gfCNCPoint1[28798] = {X 213.7862, Y 102.3021, Z -2.1667, A 0.000, B 0.000, C 0.000 }
gfCNCPoint1[28799] = {X 213.3966, Y 102.2485, Z -2.1667, A 0.000, B 0.000, C 0.000 }
gfCNCPoint1[28800] = {X 213.0070, Y 102.3021, Z -2.1667, A 0.000, B 0.000, C 0.000 }
gfCNCPoint1[28801] = {X 212.6141, Y 102.3200, Z -2.1667, A 0.000, B 0.000, C 0.000 }
gfCNCPoint1[28802] = {X 194.9870, Y 102.3200, Z -2.1667, A 0.000, B 0.000, C 0.000 }
gfCNCPoint1[28803] = {X 194.0257, Y 102.2117, Z -2.1667, A 0.000, B 0.000, C 0.000 }
gfCNCPoint1[28804] = {X 193.1126, Y 101.8922, Z -2.1667, A 0.000, B 0.000, C 0.000 }
gfCNCPoint1[28805] = {X 192.2935, Y 101.3775, Z -2.1667, A 0.000, B 0.000, C 0.000 }
gfCNCPoint1[28806] = {X 191.6094, Y 100.6935, Z -2.1667, A 0.000, B 0.000, C 0.000 }
gfCNCPoint1[28807] = {X 191.0948, Y 99.8744, Z -2.1667, A 0.000, B 0.000, C 0.000 }
gfCNCPoint1[28808] = {X 190.7753, Y 98.9613, Z -2.1667, A 0.000, B 0.000, C 0.000 }
gfCNCPoint1[28809] = {X 190.6670, Y 98.0000, Z -2.1667, A 0.000, B 0.000, C 0.000 }
gfCNCPoint1[28810] = {X 190.6670, Y 97.0659, Z -2.1667, A 0.000, B 0.000, C 0.000 }
gfCNCPoint1[28811] = {X 190.7727, Y 96.1162, Z -2.1667, A 0.000, B 0.000, C 0.000 }
gfCNCPoint1[28812] = {X 191.0846, Y 95.2129, Z -2.1667, A 0.000, B 0.000, C 0.000 }
gfCNCPoint1[28813] = {X 191.5874, Y 94.4003, Z -2.1667, A 0.000, B 0.000, C 0.000 }
gfCNCPoint1[28814] = {X 188.5647, Y 91.1002, Z -2.1667, A 0.000, B 0.000, C 0.000 }
gfCNCPoint1[28815] = {X 150.0898, Y 91.1002, Z -2.1667, A 0.000, B 0.000, C 0.000 }
gfCNCPoint1[28816] = {X 147.1445, Y 94.3633, Z -2.1667, A 0.000, B 0.000, C 0.000 }
gfCNCPoint1[28817] = {X 147.6631, Y 95.1844, Z -2.1667, A 0.000, B 0.000, C 0.000 }
gfCNCPoint1[28818] = {X 147.9867, Y 96.1001, Z -2.1667, A 0.000, B 0.000, C 0.000 }
gfCNCPoint1[28819] = {X 148.0991, Y 97.0648, Z -2.1667, A 0.000, B 0.000, C 0.000 }
gfCNCPoint1[28820] = {X 148.0991, Y 98.0000, Z -2.1667, A 0.000, B 0.000, C 0.000 }
gfCNCPoint1[28821] = {X 147.9908, Y 98.9613, Z -2.1667, A 0.000, B 0.000, C 0.000 }
gfCNCPoint1[28822] = {X 147.6713, Y 99.8744, Z -2.1667, A 0.000, B 0.000, C 0.000 }
gfCNCPoint1[28823] = {X 147.1566, Y 100.6935, Z -2.1667, A 0.000, B 0.000, C 0.000 }
gfCNCPoint1[28824] = {X 146.4726, Y 101.3775, Z -2.1667, A 0.000, B 0.000, C 0.000 }
gfCNCPoint1[28825] = {X 145.6535, Y 101.8922, Z -2.1667, A 0.000, B 0.000, C 0.000 }
gfCNCPoint1[28826] = {X 144.7404, Y 102.2117, Z -2.1667, A 0.000, B 0.000, C 0.000 }
gfCNCPoint1[28827] = {X 143.7791, Y 102.3200, Z -2.1667, A 0.000, B 0.000, C 0.000 }
gfCNCPoint1[28828] = {X 125.0000, Y 102.3200, Z -2.1667, A 0.000, B 0.000, C 0.000 }
gfCNCPoint1[28829] = {X 124.0387, Y 102.2117, Z -2.1667, A 0.000, B 0.000, C 0.000 }
gfCNCPoint1[28830] = {X 123.1256, Y 101.8922, Z -2.1667, A 0.000, B 0.000, C 0.000 }
gfCNCPoint1[28831] = {X 122.3065, Y 101.3775, Z -2.1667, A 0.000, B 0.000, C 0.000 }
gfCNCPoint1[28832] = {X 121.6225, Y 100.6935, Z -2.1667, A 0.000, B 0.000, C 0.000 }
gfCNCPoint1[28833] = {X 121.1078, Y 99.8744, Z -2.1667, A 0.000, B 0.000, C 0.000 }
gfCNCPoint1[28834] = {X 120.7883, Y 98.9613, Z -2.1667, A 0.000, B 0.000, C 0.000 }
gfCNCPoint1[28835] = {X 120.6800, Y 98.0000, Z -2.1667, A 0.000, B 0.000, C 0.000 }
gfCNCPoint1[28836] = {X 120.6800, Y 97.0659, Z -2.1667, A 0.000, B 0.000, C 0.000 }
gfCNCPoint1[28837] = {X 120.7833, Y 96.1270, Z -2.1667, A 0.000, B 0.000, C 0.000 }
gfCNCPoint1[28838] = {X 121.0882, Y 95.2329, Z -2.1667, A 0.000, B 0.000, C 0.000 }
gfCNCPoint1[28839] = {X 121.5801, Y 94.4265, Z -2.1667, A 0.000, B 0.000, C 0.000 }
gfCNCPoint1[28840] = {X 122.2355, Y 93.7463, Z -2.1667, A 0.000, B 0.000, C 0.000 }
gfCNCPoint1[28841] = {X 123.0231, Y 93.2248, Z -2.1667, A 0.000, B 0.000, C 0.000 }
gfCNCPoint1[28842] = {X 123.9052, Y 92.8870, Z -2.1667, A 0.000, B 0.000, C 0.000 }
gfCNCPoint1[28843] = {X 124.8397, Y 92.7489, Z -2.1667, A 0.000, B 0.000, C 0.000 }
gfCNCPoint1[28844] = {X 124.8829, Y 92.7325, Z -2.1667, A 0.000, B 0.000, C 0.000 }
gfCNCPoint1[28845] = {X 124.9280, Y 92.7225, Z -2.1667, A 0.000, B 0.000, C 0.000 }
gfCNCPoint1[28846] = {X 125.4501, Y 92.6450, Z -2.1667, A 0.000, B 0.000, C 0.000 }
gfCNCPoint1[28847] = {X 126.2811, Y 92.5043, Z -2.1667, A 0.000, B 0.000, C 0.000 }
gfCNCPoint1[28848] = {X 127.1008, Y 92.3085, Z -2.1667, A 0.000, B 0.000, C 0.000 }
gfCNCPoint1[28849] = {X 128.3225, Y 91.1566, Z -2.1667, A 0.000, B 0.000, C 0.000 }
gfCNCPoint1[28850] = {X 129.4799, Y 89.9402, Z -2.1667, A 0.000, B 0.000, C 0.000 }
gfCNCPoint1[28851] = {X 140.6805, Y 77.6405, Z -2.1667, A 0.000, B 0.000, C 0.000 }
gfCNCPoint1[28852] = {X 137.7230, Y 74.9473, Z -2.1667, A 0.000, B 0.000, C 0.000 }
gfCNCPoint1[28853] = {X 140.7396, Y 77.6944, Z -2.1667, A 0.000, B 0.000, C 0.000 }
gfCNCPoint1[28854] = {X 155.7331, Y 61.2296, Z -2.1667, A 0.000, B 0.000, C 0.000 }
gfCNCPoint1[28855] = {X 155.3670, Y 60.5231, Z -2.1667, A 0.000, B 0.000, C 0.000 }
gfCNCPoint1[28856] = {X 155.1393, Y 59.7606, Z -2.1667, A 0.000, B 0.000, C 0.000 }
gfCNCPoint1[28857] = {X 155.0581, Y 58.9691, Z -2.1667, A 0.000, B 0.000, C 0.000 }
gfCNCPoint1[28858] = {X 155.0580, Y 58.0000, Z -2.1667, A 0.000, B 0.000, C 0.000 }
gfCNCPoint1[28859] = {X 155.1643, Y 57.0565, Z -2.1667, A 0.000, B 0.000, C 0.000 }
gfCNCPoint1[28860] = {X 155.4778, Y 56.1603, Z -2.1667, A 0.000, B 0.000, C 0.000 }
gfCNCPoint1[28861] = {X 155.9830, Y 55.3564, Z -2.1667, A 0.000, B 0.000, C 0.000 }
gfCNCPoint1[28862] = {X 156.6544, Y 54.6850, Z -2.1667, A 0.000, B 0.000, C 0.000 }
gfCNCPoint1[28863] = {X 157.4583, Y 54.1799, Z -2.1667, A 0.000, B 0.000, C 0.000 }
gfCNCPoint1[28864] = {X 158.3545, Y 53.8663, Z -2.1667, A 0.000, B 0.000, C 0.000 }
gfCNCPoint1[28865] = {X 159.2980, Y 53.7600, Z -2.1667, A 0.000, B 0.000, C 0.000 }
gfCNCPoint1[28866] = {X 178.5335, Y 53.7600, Z -2.1667, A 0.000, B 0.000, C 0.000 }
gfCNCPoint1[28867] = {X 179.4770, Y 53.8663, Z -2.1667, A 0.000, B 0.000, C 0.000 }
gfCNCPoint1[28868] = {X 180.3732, Y 54.1799, Z -2.1667, A 0.000, B 0.000, C 0.000 }
gfCNCPoint1[28869] = {X 181.1771, Y 54.6850, Z -2.1667, A 0.000, B 0.000, C 0.000 }
gfCNCPoint1[28870] = {X 181.8485, Y 55.3564, Z -2.1667, A 0.000, B 0.000, C 0.000 }
gfCNCPoint1[28871] = {X 182.3536, Y 56.1603, Z -2.1667, A 0.000, B 0.000, C 0.000 }
gfCNCPoint1[28872] = {X 182.6672, Y 57.0565, Z -2.1667, A 0.000, B 0.000, C 0.000 }
gfCNCPoint1[28873] = {X 182.7735, Y 58.0000, Z -2.1667, A 0.000, B 0.000, C 0.000 }
gfCNCPoint1[28874] = {X 182.7735, Y 58.9342, Z -2.1667, A 0.000, B 0.000, C 0.000 }
gfCNCPoint1[28875] = {X 182.6984, Y 59.7287, Z -2.1667, A 0.000, B 0.000, C 0.000 }
gfCNCPoint1[28876] = {X 182.4757, Y 60.4950, Z -2.1667, A 0.000, B 0.000, C 0.000 }
gfCNCPoint1[28877] = {X 182.1134, Y 61.2060, Z -2.1667, A 0.000, B 0.000, C 0.000 }
gfCNCPoint1[28878] = {X 209.4186, Y 91.0079, Z -2.1667, A 0.000, B 0.000, C 0.000 }
gfCNCPoint1[28879] = {X 210.0808, Y 91.6798, Z -2.1667, A 0.000, B 0.000, C 0.000 }
gfCNCPoint1[28880] = {X 210.7901, Y 92.3017, Z -2.1667, A 0.000, B 0.000, C 0.000 }
gfCNCPoint1[28881] = {X 211.0808, Y 92.4854, Z -2.1667, A 0.000, B 0.000, C 0.000 }
gfCNCPoint1[28882] = {X 211.4066, Y 92.5950, Z -2.1667, A 0.000, B 0.000, C 0.000 }
gfCNCPoint1[28883] = {X 213.4016, Y 92.9061, Z -2.1667, A 0.000, B 0.000, C 0.000 }
gfCNCPoint1[28884] = {X 214.4545, Y 92.8170, Z -2.1667, A 0.000, B 0.000, C 0.000 }
gfCNCPoint1[28885] = {X 215.5096, Y 92.7565, Z -2.1667, A 0.000, B 0.000, C 0.000 }
gfCNCPoint1[28886] = {X 216.1940, Y 92.6814, Z -2.1667, A 0.000, B 0.000, C 0.000 }
gfCNCPoint1[28887] = {X 216.8530, Y 92.4820, Z -2.1667, A 0.000, B 0.000, C 0.000 }
gfCNCPoint1[28888] = {X 217.4644, Y 92.1653, Z -2.1667, A 0.000, B 0.000, C 0.000 }
gfCNCPoint1[28889] = {X 223.0046, Y 88.5899, Z -2.1667, A 0.000, B 0.000, C 0.000 }
gfCNCPoint1[28890] = {X 246.0044, Y 73.8823, Z -2.1667, A 0.000, B 0.000, C 0.000 }
gfCNCPoint1[28891] = {X 221.6602, Y 64.3284, Z -2.1667, A 0.000, B 0.000, C 0.000 }
gfCNCPoint1[28892] = {X 219.8842, Y 63.7340, Z -2.1667, A 0.000, B 0.000, C 0.000 }
gfCNCPoint1[28893] = {X 218.0518, Y 63.3467, Z -2.1667, A 0.000, B 0.000, C 0.000 }
gfCNCPoint1[28894] = {X 216.1871, Y 63.1716, Z -2.1667, A 0.000, B 0.000, C 0.000 }
gfCNCPoint1[28895] = {X 215.2725, Y 63.0399, Z -2.1667, A 0.000, B 0.000, C 0.000 }
gfCNCPoint1[28896] = {X 214.4081, Y 62.7131, Z -2.1667, A 0.000, B 0.000, C 0.000 }
gfCNCPoint1[28897] = {X 213.6351, Y 62.2068, Z -2.1667, A 0.000, B 0.000, C 0.000 }
gfCNCPoint1[28898] = {X 212.9901, Y 61.5450, Z -2.1667, A 0.000, B 0.000, C 0.000 }
gfCNCPoint1[28899] = {X 212.5038, Y 60.7593, Z -2.1667, A 0.000, B 0.000, C 0.000 }
gfCNCPoint1[28900] = {X 212.1992, Y 59.8868, Z -2.1667, A 0.000, B 0.000, C 0.000 }
gfCNCPoint1[28901] = {X 212.0910, Y 58.9691, Z -2.1667, A 0.000, B 0.000, C 0.000 }
gfCNCPoint1[28902] = {X 212.0908, Y 58.0000, Z -2.1667, A 0.000, B 0.000, C 0.000 }
gfCNCPoint1[28903] = {X 212.1971, Y 57.0565, Z -2.1667, A 0.000, B 0.000, C 0.000 }
gfCNCPoint1[28904] = {X 212.5107, Y 56.1603, Z -2.1667, A 0.000, B 0.000, C 0.000 }
gfCNCPoint1[28905] = {X 213.0158, Y 55.3564, Z -2.1667, A 0.000, B 0.000, C 0.000 }
gfCNCPoint1[28906] = {X 213.6872, Y 54.6850, Z -2.1667, A 0.000, B 0.000, C 0.000 }
gfCNCPoint1[28907] = {X 214.4911, Y 54.1799, Z -2.1667, A 0.000, B 0.000, C 0.000 }
gfCNCPoint1[28908] = {X 215.3873, Y 53.8663, Z -2.1667, A 0.000, B 0.000, C 0.000 }
gfCNCPoint1[28909] = {X 216.3308, Y 53.7600, Z -2.1667, A 0.000, B 0.000, C 0.000 }
gfCNCPoint1[28910] = {X 237.2617, Y 53.7600, Z -2.1667, A 0.000, B 0.000, C 0.000 }
gfCNCPoint1[28911] = {X 238.2052, Y 53.8663, Z -2.1667, A 0.000, B 0.000, C 0.000 }
gfCNCPoint1[28912] = {X 239.1014, Y 54.1799, Z -2.1667, A 0.000, B 0.000, C 0.000 }
gfCNCPoint1[28913] = {X 239.9053, Y 54.6850, Z -2.1667, A 0.000, B 0.000, C 0.000 }
gfCNCPoint1[28914] = {X 240.5767, Y 55.3564, Z -2.1667, A 0.000, B 0.000, C 0.000 }
gfCNCPoint1[28915] = {X 241.0818, Y 56.1603, Z -2.1667, A 0.000, B 0.000, C 0.000 }
gfCNCPoint1[28916] = {X 241.3954, Y 57.0565, Z -2.1667, A 0.000, B 0.000, C 0.000 }
gfCNCPoint1[28917] = {X 241.5017, Y 58.0000, Z -2.1667, A 0.000, B 0.000, C 0.000 }
gfCNCPoint1[28918] = {X 241.5017, Y 58.2875, Z -2.1667, A 0.000, B 0.000, C 0.000 }
gfCNCPoint1[28919] = {X 247.4591, Y 60.6101, Z -2.1667, A 0.000, B 0.000, C 0.000 }
gfCNCPoint1[28920] = {X 275.7138, Y 71.8208, Z -2.1667, A 0.000, B 0.000, C 0.000 }
gfCNCPoint1[28921] = {X 275.7145, Y 63.1423, Z -2.1667, A 0.000, B 0.000, C 0.000 }
gfCNCPoint1[28922] = {X 274.8658, Y 62.9477, Z -2.1667, A 0.000, B 0.000, C 0.000 }
gfCNCPoint1[28923] = {X 274.0748, Y 62.5838, Z -2.1667, A 0.000, B 0.000, C 0.000 }
gfCNCPoint1[28924] = {X 273.3747, Y 62.0661, Z -2.1667, A 0.000, B 0.000, C 0.000 }
gfCNCPoint1[28925] = {X 272.7952, Y 61.4163, Z -2.1667, A 0.000, B 0.000, C 0.000 }
gfCNCPoint1[28926] = {X 272.3607, Y 60.6618, Z -2.1667, A 0.000, B 0.000, C 0.000 }
gfCNCPoint1[28927] = {X 272.0894, Y 59.8344, Z -2.1667, A 0.000, B 0.000, C 0.000 }
gfCNCPoint1[28928] = {X 271.9928, Y 58.9691, Z -2.1667, A 0.000, B 0.000, C 0.000 }
gfCNCPoint1[28929] = {X 271.9927, Y 58.0000, Z -2.1667, A 0.000, B 0.000, C 0.000 }
gfCNCPoint1[28930] = {X 272.0990, Y 57.0565, Z -2.1667, A 0.000, B 0.000, C 0.000 }
gfCNCPoint1[28931] = {X 272.4126, Y 56.1603, Z -2.1667, A 0.000, B 0.000, C 0.000 }
gfCNCPoint1[28932] = {X 272.9177, Y 55.3564, Z -2.1667, A 0.000, B 0.000, C 0.000 }
gfCNCPoint1[28933] = {X 273.5891, Y 54.6850, Z -2.1667, A 0.000, B 0.000, C 0.000 }
gfCNCPoint1[28934] = {X 274.3930, Y 54.1799, Z -2.1667, A 0.000, B 0.000, C 0.000 }
gfCNCPoint1[28935] = {X 275.2892, Y 53.8663, Z -2.1667, A 0.000, B 0.000, C 0.000 }
gfCNCPoint1[28936] = {X 276.2327, Y 53.7600, Z -2.1667, A 0.000, B 0.000, C 0.000 }
gfCNCPoint1[28937] = {X 292.7731, Y 53.7600, Z -2.1667, A 0.000, B 0.000, C 0.000 }
gfCNCPoint1[28938] = {X 293.7166, Y 53.8663, Z -2.1667, A 0.000, B 0.000, C 0.000 }
gfCNCPoint1[28939] = {X 294.6128, Y 54.1799, Z -2.1667, A 0.000, B 0.000, C 0.000 }
gfCNCPoint1[28940] = {X 295.4167, Y 54.6850, Z -2.1667, A 0.000, B 0.000, C 0.000 }
gfCNCPoint1[28941] = {X 296.0881, Y 55.3564, Z -2.1667, A 0.000, B 0.000, C 0.000 }
gfCNCPoint1[28942] = {X 296.5932, Y 56.1603, Z -2.1667, A 0.000, B 0.000, C 0.000 }
gfCNCPoint1[28943] = {X 296.9068, Y 57.0565, Z -2.1667, A 0.000, B 0.000, C 0.000 }
gfCNCPoint1[28944] = {X 297.0131, Y 58.0000, Z -2.1667, A 0.000, B 0.000, C 0.000 }
gfCNCPoint1[28945] = {X 297.0131, Y 58.9349, Z -2.1667, A 0.000, B 0.000, C 0.000 }
gfCNCPoint1[28946] = {X 296.8928, Y 59.9252, Z -2.1667, A 0.000, B 0.000, C 0.000 }
gfCNCPoint1[28947] = {X 296.5453, Y 60.8602, Z -2.1667, A 0.000, B 0.000, C 0.000 }
gfCNCPoint1[28948] = {X 295.9899, Y 61.6887, Z -2.1667, A 0.000, B 0.000, C 0.000 }
gfCNCPoint1[28949] = {X 295.2568, Y 62.3652, Z -2.1667, A 0.000, B 0.000, C 0.000 }
gfCNCPoint1[28950] = {X 294.3864, Y 62.8526, Z -2.1667, A 0.000, B 0.000, C 0.000 }
gfCNCPoint1[28951] = {X 293.4266, Y 63.1240, Z -2.1667, A 0.000, B 0.000, C 0.000 }
gfCNCPoint1[28952] = {X 293.2918, Y 63.1662, Z -2.1667, A 0.000, B 0.000, C 0.000 }
gfCNCPoint1[28953] = {X 293.3041, Y 92.8516, Z -2.1667, A 0.000, B 0.000, C 0.000 }
gfCNCPoint1[28954] = {X 294.1535, Y 93.0547, Z -2.1667, A 0.000, B 0.000, C 0.000 }
gfCNCPoint1[28955] = {X 294.9439, Y 93.4263, Z -2.1667, A 0.000, B 0.000, C 0.000 }
gfCNCPoint1[28956] = {X 295.6421, Y 93.9508, Z -2.1667, A 0.000, B 0.000, C 0.000 }
gfCNCPoint1[28957] = {X 296.2192, Y 94.6063, Z -2.1667, A 0.000, B 0.000, C 0.000 }
gfCNCPoint1[28958] = {X 296.6509, Y 95.3655, Z -2.1667, A 0.000, B 0.000, C 0.000 }
gfCNCPoint1[28959] = {X 296.9193, Y 96.1966, Z -2.1667, A 0.000, B 0.000, C 0.000 }
gfCNCPoint1[28960] = {X 297.0131, Y 97.0649, Z -2.1667, A 0.000, B 0.000, C 0.000 }
gfCNCPoint1[28961] = {X 297.0131, Y 98.0000, Z -2.1667, A 0.000, B 0.000, C 0.000 }
gfCNCPoint1[28962] = {X 296.9068, Y 98.9435, Z -2.1667, A 0.000, B 0.000, C 0.000 }
gfCNCPoint1[28963] = {X 296.5932, Y 99.8397, Z -2.1667, A 0.000, B 0.000, C 0.000 }
gfCNCPoint1[28964] = {X 296.0881, Y 100.6436, Z -2.1667, A 0.000, B 0.000, C 0.000 }
gfCNCPoint1[28965] = {X 295.4167, Y 101.3150, Z -2.1667, A 0.000, B 0.000, C 0.000 }
gfCNCPoint1[28966] = {X 294.6128, Y 101.8201, Z -2.1667, A 0.000, B 0.000, C 0.000 }
gfCNCPoint1[28967] = {X 293.7166, Y 102.1337, Z -2.1667, A 0.000, B 0.000, C 0.000 }
gfCNCPoint1[28968] = {X 292.7731, Y 102.2400, Z -2.1667, A 0.000, B 0.000, C 0.000 }
gfCNCPoint1[28969] = {X 276.2327, Y 102.2400, Z -2.1667, A 0.000, B 0.000, C 0.000 }
gfCNCPoint1[28970] = {X 275.2892, Y 102.1337, Z -2.1667, A 0.000, B 0.000, C 0.000 }
gfCNCPoint1[28971] = {X 274.3930, Y 101.8201, Z -2.1667, A 0.000, B 0.000, C 0.000 }
gfCNCPoint1[28972] = {X 273.5891, Y 101.3150, Z -2.1667, A 0.000, B 0.000, C 0.000 }
gfCNCPoint1[28973] = {X 272.9177, Y 100.6436, Z -2.1667, A 0.000, B 0.000, C 0.000 }
gfCNCPoint1[28974] = {X 272.4126, Y 99.8397, Z -2.1667, A 0.000, B 0.000, C 0.000 }
gfCNCPoint1[28975] = {X 272.0990, Y 98.9435, Z -2.1667, A 0.000, B 0.000, C 0.000 }
gfCNCPoint1[28976] = {X 271.9927, Y 98.0000, Z -2.1667, A 0.000, B 0.000, C 0.000 }
gfCNCPoint1[28977] = {X 271.9927, Y 97.0659, Z -2.1667, A 0.000, B 0.000, C 0.000 }
gfCNCPoint1[28978] = {X 272.0830, Y 96.1957, Z -2.1667, A 0.000, B 0.000, C 0.000 }
gfCNCPoint1[28979] = {X 272.3499, Y 95.3624, Z -2.1667, A 0.000, B 0.000, C 0.000 }
gfCNCPoint1[28980] = {X 272.7823, Y 94.6018, Z -2.1667, A 0.000, B 0.000, C 0.000 }
gfCNCPoint1[28981] = {X 273.3615, Y 93.9460, Z -2.1667, A 0.000, B 0.000, C 0.000 }
gfCNCPoint1[28982] = {X 274.0630, Y 93.4231, Z -2.1667, A 0.000, B 0.000, C 0.000 }
gfCNCPoint1[28983] = {X 274.8569, Y 93.0553, Z -2.1667, A 0.000, B 0.000, C 0.000 }
gfCNCPoint1[28984] = {X 275.7094, Y 92.8584, Z -2.1667, A 0.000, B 0.000, C 0.000 }
gfCNCPoint1[28985] = {X 275.7094, Y 85.5404, Z -2.1667, A 0.000, B 0.000, C 0.000 }
gfCNCPoint1[28986] = {X 262.6311, Y 80.4137, Z -2.1667, A 0.000, B 0.000, C 0.000 }
gfCNCPoint1[28987] = {X 262.2329, Y 80.6642, Z -2.1667, A 0.000, B 0.000, C 0.000 }
gfCNCPoint1[28988] = {X 237.7156, Y 96.5447, Z -2.1667, A 0.000, B 0.000, C 0.000 }
gfCNCPoint1[28989] = {X 237.7198, Y 97.0649, Z -2.1667, A 0.000, B 0.000, C 0.000 }
gfCNCPoint1[28990] = {X 237.7198, Y 98.0000, Z -2.1667, A 0.000, B 0.000, C 0.000 }
gfCNCPoint1[28991] = {X 237.6135, Y 98.9435, Z -2.1667, A 0.000, B 0.000, C 0.000 }
gfCNCPoint1[28992] = {X 237.2999, Y 99.8397, Z -2.1667, A 0.000, B 0.000, C 0.000 }
gfCNCPoint1[28993] = {X 236.7948, Y 100.6436, Z -2.1667, A 0.000, B 0.000, C 0.000 }
gfCNCPoint1[28994] = {X 236.1234, Y 101.3150, Z -2.1667, A 0.000, B 0.000, C 0.000 }
gfCNCPoint1[28995] = {X 235.3195, Y 101.8201, Z -2.1667, A 0.000, B 0.000, C 0.000 }
gfCNCPoint1[28996] = {X 234.4233, Y 102.1337, Z -2.1667, A 0.000, B 0.000, C 0.000 }
gfCNCPoint1[28997] = {X 233.4798, Y 102.2400, Z -2.1667, A 0.000, B 0.000, C 0.000 }
gfCNCPoint1[28998] = {X 214.1790, Y 102.2400, Z -2.1667, A 0.000, B 0.000, C 0.000 }
gfCNCPoint1[28999] = {X 213.7861, Y 102.2218, Z -2.1667, A 0.000, B 0.000, C 0.000 }
gfCNCPoint1[29000] = {X 213.3966, Y 102.1672, Z -2.1667, A 0.000, B 0.000, C 0.000 }
gfCNCPoint1[29001] = {X 213.0070, Y 102.2218, Z -2.1667, A 0.000, B 0.000, C 0.000 }
gfCNCPoint1[29002] = {X 212.6141, Y 102.2400, Z -2.1667, A 0.000, B 0.000, C 0.000 }
gfCNCPoint1[29003] = {X 194.9870, Y 102.2400, Z -2.1667, A 0.000, B 0.000, C 0.000 }
gfCNCPoint1[29004] = {X 194.0435, Y 102.1337, Z -2.1667, A 0.000, B 0.000, C 0.000 }
gfCNCPoint1[29005] = {X 193.1473, Y 101.8201, Z -2.1667, A 0.000, B 0.000, C 0.000 }
gfCNCPoint1[29006] = {X 192.3434, Y 101.3150, Z -2.1667, A 0.000, B 0.000, C 0.000 }
gfCNCPoint1[29007] = {X 191.6720, Y 100.6436, Z -2.1667, A 0.000, B 0.000, C 0.000 }
gfCNCPoint1[29008] = {X 191.1669, Y 99.8397, Z -2.1667, A 0.000, B 0.000, C 0.000 }
gfCNCPoint1[29009] = {X 190.8533, Y 98.9435, Z -2.1667, A 0.000, B 0.000, C 0.000 }
gfCNCPoint1[29010] = {X 190.7470, Y 98.0000, Z -2.1667, A 0.000, B 0.000, C 0.000 }
gfCNCPoint1[29011] = {X 190.7470, Y 97.0659, Z -2.1667, A 0.000, B 0.000, C 0.000 }
gfCNCPoint1[29012] = {X 190.8557, Y 96.1118, Z -2.1667, A 0.000, B 0.000, C 0.000 }
gfCNCPoint1[29013] = {X 191.1764, Y 95.2065, Z -2.1667, A 0.000, B 0.000, C 0.000 }
gfCNCPoint1[29014] = {X 191.6926, Y 94.3967, Z -2.1667, A 0.000, B 0.000, C 0.000 }
gfCNCPoint1[29015] = {X 188.5999, Y 91.0202, Z -2.1667, A 0.000, B 0.000, C 0.000 }
gfCNCPoint1[29016] = {X 150.0543, Y 91.0202, Z -2.1667, A 0.000, B 0.000, C 0.000 }
gfCNCPoint1[29017] = {X 147.0391, Y 94.3606, Z -2.1667, A 0.000, B 0.000, C 0.000 }
gfCNCPoint1[29018] = {X 147.5712, Y 95.1787, Z -2.1667, A 0.000, B 0.000, C 0.000 }
gfCNCPoint1[29019] = {X 147.9036, Y 96.0961, Z -2.1667, A 0.000, B 0.000, C 0.000 }
gfCNCPoint1[29020] = {X 148.0191, Y 97.0651, Z -2.1667, A 0.000, B 0.000, C 0.000 }
gfCNCPoint1[29021] = {X 148.0191, Y 98.0000, Z -2.1667, A 0.000, B 0.000, C 0.000 }
gfCNCPoint1[29022] = {X 147.9128, Y 98.9435, Z -2.1667, A 0.000, B 0.000, C 0.000 }
gfCNCPoint1[29023] = {X 147.5992, Y 99.8397, Z -2.1667, A 0.000, B 0.000, C 0.000 }
gfCNCPoint1[29024] = {X 147.0941, Y 100.6436, Z -2.1667, A 0.000, B 0.000, C 0.000 }
gfCNCPoint1[29025] = {X 146.4227, Y 101.3150, Z -2.1667, A 0.000, B 0.000, C 0.000 }
gfCNCPoint1[29026] = {X 145.6188, Y 101.8201, Z -2.1667, A 0.000, B 0.000, C 0.000 }
gfCNCPoint1[29027] = {X 144.7226, Y 102.1337, Z -2.1667, A 0.000, B 0.000, C 0.000 }
gfCNCPoint1[29028] = {X 143.7791, Y 102.2400, Z -2.1667, A 0.000, B 0.000, C 0.000 }
gfCNCPoint1[29029] = {X 125.0000, Y 102.2400, Z -2.1667, A 0.000, B 0.000, C 0.000 }
gfCNCPoint1[29030] = {X 124.0565, Y 102.1337, Z -2.1667, A 0.000, B 0.000, C 0.000 }
gfCNCPoint1[29031] = {X 123.1603, Y 101.8201, Z -2.1667, A 0.000, B 0.000, C 0.000 }
gfCNCPoint1[29032] = {X 122.3564, Y 101.3150, Z -2.1667, A 0.000, B 0.000, C 0.000 }
gfCNCPoint1[29033] = {X 121.6850, Y 100.6436, Z -2.1667, A 0.000, B 0.000, C 0.000 }
gfCNCPoint1[29034] = {X 121.1799, Y 99.8397, Z -2.1667, A 0.000, B 0.000, C 0.000 }
gfCNCPoint1[29035] = {X 120.8663, Y 98.9435, Z -2.1667, A 0.000, B 0.000, C 0.000 }
gfCNCPoint1[29036] = {X 120.7600, Y 98.0000, Z -2.1667, A 0.000, B 0.000, C 0.000 }
gfCNCPoint1[29037] = {X 120.7600, Y 97.0659, Z -2.1667, A 0.000, B 0.000, C 0.000 }
gfCNCPoint1[29038] = {X 120.8619, Y 96.1420, Z -2.1667, A 0.000, B 0.000, C 0.000 }
gfCNCPoint1[29039] = {X 121.1627, Y 95.2624, Z -2.1667, A 0.000, B 0.000, C 0.000 }
gfCNCPoint1[29040] = {X 121.6479, Y 94.4695, Z -2.1667, A 0.000, B 0.000, C 0.000 }
gfCNCPoint1[29041] = {X 122.2943, Y 93.8015, Z -2.1667, A 0.000, B 0.000, C 0.000 }
gfCNCPoint1[29042] = {X 123.0707, Y 93.2903, Z -2.1667, A 0.000, B 0.000, C 0.000 }
gfCNCPoint1[29043] = {X 123.9398, Y 92.9606, Z -2.1667, A 0.000, B 0.000, C 0.000 }
gfCNCPoint1[29044] = {X 124.8599, Y 92.8282, Z -2.1667, A 0.000, B 0.000, C 0.000 }
gfCNCPoint1[29045] = {X 124.8987, Y 92.8114, Z -2.1667, A 0.000, B 0.000, C 0.000 }
gfCNCPoint1[29046] = {X 124.9397, Y 92.8016, Z -2.1667, A 0.000, B 0.000, C 0.000 }
gfCNCPoint1[29047] = {X 125.4608, Y 92.7243, Z -2.1667, A 0.000, B 0.000, C 0.000 }
gfCNCPoint1[29048] = {X 126.3063, Y 92.5808, Z -2.1667, A 0.000, B 0.000, C 0.000 }
gfCNCPoint1[29049] = {X 127.1401, Y 92.3807, Z -2.1667, A 0.000, B 0.000, C 0.000 }
gfCNCPoint1[29050] = {X 128.3723, Y 91.2199, Z -2.1667, A 0.000, B 0.000, C 0.000 }
gfCNCPoint1[29051] = {X 129.5394, Y 89.9938, Z -2.1667, A 0.000, B 0.000, C 0.000 }
gfCNCPoint1[29052] = {X 140.7396, Y 77.6944, Z -2.1667, A 0.000, B 0.000, C 0.000 }
gfCNCPoint1[29053] = {X 137.7821, Y 75.0012, Z -2.1667, A 0.000, B 0.000, C 0.000 }
gfCNCPoint1[29054] = {X 140.7988, Y 77.7483, Z -2.1667, A 0.000, B 0.000, C 0.000 }
gfCNCPoint1[29055] = {X 155.8340, Y 61.2376, Z -2.1667, A 0.000, B 0.000, C 0.000 }
gfCNCPoint1[29056] = {X 155.4567, Y 60.5310, Z -2.1667, A 0.000, B 0.000, C 0.000 }
gfCNCPoint1[29057] = {X 155.2218, Y 59.7651, Z -2.1667, A 0.000, B 0.000, C 0.000 }
gfCNCPoint1[29058] = {X 155.1381, Y 58.9684, Z -2.1667, A 0.000, B 0.000, C 0.000 }
gfCNCPoint1[29059] = {X 155.1380, Y 58.0000, Z -2.1667, A 0.000, B 0.000, C 0.000 }
gfCNCPoint1[29060] = {X 155.2423, Y 57.0743, Z -2.1667, A 0.000, B 0.000, C 0.000 }
gfCNCPoint1[29061] = {X 155.5499, Y 56.1950, Z -2.1667, A 0.000, B 0.000, C 0.000 }
gfCNCPoint1[29062] = {X 156.0455, Y 55.4063, Z -2.1667, A 0.000, B 0.000, C 0.000 }
gfCNCPoint1[29063] = {X 156.7042, Y 54.7476, Z -2.1667, A 0.000, B 0.000, C 0.000 }
gfCNCPoint1[29064] = {X 157.4930, Y 54.2520, Z -2.1667, A 0.000, B 0.000, C 0.000 }
gfCNCPoint1[29065] = {X 158.3723, Y 53.9443, Z -2.1667, A 0.000, B 0.000, C 0.000 }
gfCNCPoint1[29066] = {X 159.2980, Y 53.8400, Z -2.1667, A 0.000, B 0.000, C 0.000 }
gfCNCPoint1[29067] = {X 178.5335, Y 53.8400, Z -2.1667, A 0.000, B 0.000, C 0.000 }
gfCNCPoint1[29068] = {X 179.4592, Y 53.9443, Z -2.1667, A 0.000, B 0.000, C 0.000 }
gfCNCPoint1[29069] = {X 180.3385, Y 54.2520, Z -2.1667, A 0.000, B 0.000, C 0.000 }
gfCNCPoint1[29070] = {X 181.1272, Y 54.7476, Z -2.1667, A 0.000, B 0.000, C 0.000 }
gfCNCPoint1[29071] = {X 181.7859, Y 55.4063, Z -2.1667, A 0.000, B 0.000, C 0.000 }
gfCNCPoint1[29072] = {X 182.2815, Y 56.1950, Z -2.1667, A 0.000, B 0.000, C 0.000 }
gfCNCPoint1[29073] = {X 182.5892, Y 57.0743, Z -2.1667, A 0.000, B 0.000, C 0.000 }
gfCNCPoint1[29074] = {X 182.6935, Y 58.0000, Z -2.1667, A 0.000, B 0.000, C 0.000 }
gfCNCPoint1[29075] = {X 182.6935, Y 58.9342, Z -2.1667, A 0.000, B 0.000, C 0.000 }
gfCNCPoint1[29076] = {X 182.6159, Y 59.7337, Z -2.1667, A 0.000, B 0.000, C 0.000 }
gfCNCPoint1[29077] = {X 182.3862, Y 60.5034, Z -2.1667, A 0.000, B 0.000, C 0.000 }
gfCNCPoint1[29078] = {X 182.0128, Y 61.2145, Z -2.1667, A 0.000, B 0.000, C 0.000 }
gfCNCPoint1[29079] = {X 209.3596, Y 91.0620, Z -2.1667, A 0.000, B 0.000, C 0.000 }
gfCNCPoint1[29080] = {X 210.0259, Y 91.7380, Z -2.1667, A 0.000, B 0.000, C 0.000 }
gfCNCPoint1[29081] = {X 210.7396, Y 92.3637, Z -2.1667, A 0.000, B 0.000, C 0.000 }
gfCNCPoint1[29082] = {X 211.0473, Y 92.5580, Z -2.1667, A 0.000, B 0.000, C 0.000 }
gfCNCPoint1[29083] = {X 211.3924, Y 92.6737, Z -2.1667, A 0.000, B 0.000, C 0.000 }
gfCNCPoint1[29084] = {X 213.3993, Y 92.9868, Z -2.1667, A 0.000, B 0.000, C 0.000 }
gfCNCPoint1[29085] = {X 214.4546, Y 92.8972, Z -2.1667, A 0.000, B 0.000, C 0.000 }
gfCNCPoint1[29086] = {X 215.5120, Y 92.8365, Z -2.1667, A 0.000, B 0.000, C 0.000 }
gfCNCPoint1[29087] = {X 216.2108, Y 92.7596, Z -2.1667, A 0.000, B 0.000, C 0.000 }
gfCNCPoint1[29088] = {X 216.8836, Y 92.5560, Z -2.1667, A 0.000, B 0.000, C 0.000 }
gfCNCPoint1[29089] = {X 217.5077, Y 92.2325, Z -2.1667, A 0.000, B 0.000, C 0.000 }
gfCNCPoint1[29090] = {X 223.0478, Y 88.6572, Z -2.1667, A 0.000, B 0.000, C 0.000 }
gfCNCPoint1[29091] = {X 246.1797, Y 73.8652, Z -2.1667, A 0.000, B 0.000, C 0.000 }
gfCNCPoint1[29092] = {X 221.6899, Y 64.2541, Z -2.1667, A 0.000, B 0.000, C 0.000 }
gfCNCPoint1[29093] = {X 219.9052, Y 63.6568, Z -2.1667, A 0.000, B 0.000, C 0.000 }
gfCNCPoint1[29094] = {X 218.0638, Y 63.2676, Z -2.1667, A 0.000, B 0.000, C 0.000 }
gfCNCPoint1[29095] = {X 216.1900, Y 63.0917, Z -2.1667, A 0.000, B 0.000, C 0.000 }
gfCNCPoint1[29096] = {X 215.2926, Y 62.9624, Z -2.1667, A 0.000, B 0.000, C 0.000 }
gfCNCPoint1[29097] = {X 214.4445, Y 62.6418, Z -2.1667, A 0.000, B 0.000, C 0.000 }
gfCNCPoint1[29098] = {X 213.6860, Y 62.1451, Z -2.1667, A 0.000, B 0.000, C 0.000 }
gfCNCPoint1[29099] = {X 213.0532, Y 61.4958, Z -2.1667, A 0.000, B 0.000, C 0.000 }
gfCNCPoint1[29100] = {X 212.5760, Y 60.7249, Z -2.1667, A 0.000, B 0.000, C 0.000 }
gfCNCPoint1[29101] = {X 212.2772, Y 59.8688, Z -2.1667, A 0.000, B 0.000, C 0.000 }
gfCNCPoint1[29102] = {X 212.1710, Y 58.9684, Z -2.1667, A 0.000, B 0.000, C 0.000 }
gfCNCPoint1[29103] = {X 212.1708, Y 58.0000, Z -2.1667, A 0.000, B 0.000, C 0.000 }
gfCNCPoint1[29104] = {X 212.2751, Y 57.0743, Z -2.1667, A 0.000, B 0.000, C 0.000 }
gfCNCPoint1[29105] = {X 212.5828, Y 56.1950, Z -2.1667, A 0.000, B 0.000, C 0.000 }
gfCNCPoint1[29106] = {X 213.0784, Y 55.4063, Z -2.1667, A 0.000, B 0.000, C 0.000 }
gfCNCPoint1[29107] = {X 213.7371, Y 54.7476, Z -2.1667, A 0.000, B 0.000, C 0.000 }
gfCNCPoint1[29108] = {X 214.5259, Y 54.2520, Z -2.1667, A 0.000, B 0.000, C 0.000 }
gfCNCPoint1[29109] = {X 215.4051, Y 53.9443, Z -2.1667, A 0.000, B 0.000, C 0.000 }
gfCNCPoint1[29110] = {X 216.3308, Y 53.8400, Z -2.1667, A 0.000, B 0.000, C 0.000 }
gfCNCPoint1[29111] = {X 237.2617, Y 53.8400, Z -2.1667, A 0.000, B 0.000, C 0.000 }
gfCNCPoint1[29112] = {X 238.1874, Y 53.9443, Z -2.1667, A 0.000, B 0.000, C 0.000 }
gfCNCPoint1[29113] = {X 239.0666, Y 54.2520, Z -2.1667, A 0.000, B 0.000, C 0.000 }
gfCNCPoint1[29114] = {X 239.8554, Y 54.7476, Z -2.1667, A 0.000, B 0.000, C 0.000 }
gfCNCPoint1[29115] = {X 240.5141, Y 55.4063, Z -2.1667, A 0.000, B 0.000, C 0.000 }
gfCNCPoint1[29116] = {X 241.0097, Y 56.1950, Z -2.1667, A 0.000, B 0.000, C 0.000 }
gfCNCPoint1[29117] = {X 241.3174, Y 57.0743, Z -2.1667, A 0.000, B 0.000, C 0.000 }
gfCNCPoint1[29118] = {X 241.4217, Y 58.0000, Z -2.1667, A 0.000, B 0.000, C 0.000 }
gfCNCPoint1[29119] = {X 241.4217, Y 58.3422, Z -2.1667, A 0.000, B 0.000, C 0.000 }
gfCNCPoint1[29120] = {X 247.4298, Y 60.6845, Z -2.1667, A 0.000, B 0.000, C 0.000 }
gfCNCPoint1[29121] = {X 275.7938, Y 71.9386, Z -2.1667, A 0.000, B 0.000, C 0.000 }
gfCNCPoint1[29122] = {X 275.7945, Y 63.0709, Z -2.1667, A 0.000, B 0.000, C 0.000 }
gfCNCPoint1[29123] = {X 275.6921, Y 63.0588, Z -2.1667, A 0.000, B 0.000, C 0.000 }
gfCNCPoint1[29124] = {X 275.5901, Y 63.0441, Z -2.1667, A 0.000, B 0.000, C 0.000 }
gfCNCPoint1[29125] = {X 274.6524, Y 62.7822, Z -2.1667, A 0.000, B 0.000, C 0.000 }
gfCNCPoint1[29126] = {X 273.8013, Y 62.3095, Z -2.1667, A 0.000, B 0.000, C 0.000 }
gfCNCPoint1[29127] = {X 273.0833, Y 61.6519, Z -2.1667, A 0.000, B 0.000, C 0.000 }
gfCNCPoint1[29128] = {X 272.5378, Y 60.8455, Z -2.1667, A 0.000, B 0.000, C 0.000 }
gfCNCPoint1[29129] = {X 272.1947, Y 59.9344, Z -2.1667, A 0.000, B 0.000, C 0.000 }
gfCNCPoint1[29130] = {X 272.0728, Y 58.9684, Z -2.1667, A 0.000, B 0.000, C 0.000 }
gfCNCPoint1[29131] = {X 272.0727, Y 58.0000, Z -2.1667, A 0.000, B 0.000, C 0.000 }
gfCNCPoint1[29132] = {X 272.1770, Y 57.0743, Z -2.1667, A 0.000, B 0.000, C 0.000 }
gfCNCPoint1[29133] = {X 272.4847, Y 56.1950, Z -2.1667, A 0.000, B 0.000, C 0.000 }
gfCNCPoint1[29134] = {X 272.9803, Y 55.4063, Z -2.1667, A 0.000, B 0.000, C 0.000 }
gfCNCPoint1[29135] = {X 273.6390, Y 54.7476, Z -2.1667, A 0.000, B 0.000, C 0.000 }
gfCNCPoint1[29136] = {X 274.4277, Y 54.2520, Z -2.1667, A 0.000, B 0.000, C 0.000 }
gfCNCPoint1[29137] = {X 275.3070, Y 53.9443, Z -2.1667, A 0.000, B 0.000, C 0.000 }
gfCNCPoint1[29138] = {X 276.2327, Y 53.8400, Z -2.1667, A 0.000, B 0.000, C 0.000 }
gfCNCPoint1[29139] = {X 292.7731, Y 53.8400, Z -2.1667, A 0.000, B 0.000, C 0.000 }
gfCNCPoint1[29140] = {X 293.6988, Y 53.9443, Z -2.1667, A 0.000, B 0.000, C 0.000 }
gfCNCPoint1[29141] = {X 294.5780, Y 54.2520, Z -2.1667, A 0.000, B 0.000, C 0.000 }
gfCNCPoint1[29142] = {X 295.3668, Y 54.7476, Z -2.1667, A 0.000, B 0.000, C 0.000 }
gfCNCPoint1[29143] = {X 296.0255, Y 55.4063, Z -2.1667, A 0.000, B 0.000, C 0.000 }
gfCNCPoint1[29144] = {X 296.5211, Y 56.1950, Z -2.1667, A 0.000, B 0.000, C 0.000 }
gfCNCPoint1[29145] = {X 296.8288, Y 57.0743, Z -2.1667, A 0.000, B 0.000, C 0.000 }
gfCNCPoint1[29146] = {X 296.9331, Y 58.0000, Z -2.1667, A 0.000, B 0.000, C 0.000 }
gfCNCPoint1[29147] = {X 296.9331, Y 58.9346, Z -2.1667, A 0.000, B 0.000, C 0.000 }
gfCNCPoint1[29148] = {X 296.8150, Y 59.9063, Z -2.1667, A 0.000, B 0.000, C 0.000 }
gfCNCPoint1[29149] = {X 296.4741, Y 60.8237, Z -2.1667, A 0.000, B 0.000, C 0.000 }
gfCNCPoint1[29150] = {X 295.9291, Y 61.6367, Z -2.1667, A 0.000, B 0.000, C 0.000 }
gfCNCPoint1[29151] = {X 295.2098, Y 62.3005, Z -2.1667, A 0.000, B 0.000, C 0.000 }
gfCNCPoint1[29152] = {X 294.3558, Y 62.7787, Z -2.1667, A 0.000, B 0.000, C 0.000 }
gfCNCPoint1[29153] = {X 293.4140, Y 63.0450, Z -2.1667, A 0.000, B 0.000, C 0.000 }
gfCNCPoint1[29154] = {X 293.3177, Y 63.0592, Z -2.1667, A 0.000, B 0.000, C 0.000 }
gfCNCPoint1[29155] = {X 293.2210, Y 63.0712, Z -2.1667, A 0.000, B 0.000, C 0.000 }
gfCNCPoint1[29156] = {X 293.2118, Y 63.1622, Z -2.1667, A 0.000, B 0.000, C 0.000 }
gfCNCPoint1[29157] = {X 293.2242, Y 92.9222, Z -2.1667, A 0.000, B 0.000, C 0.000 }
gfCNCPoint1[29158] = {X 293.3189, Y 92.9343, Z -2.1667, A 0.000, B 0.000, C 0.000 }
gfCNCPoint1[29159] = {X 293.4132, Y 92.9486, Z -2.1667, A 0.000, B 0.000, C 0.000 }
gfCNCPoint1[29160] = {X 294.3547, Y 93.2175, Z -2.1667, A 0.000, B 0.000, C 0.000 }
gfCNCPoint1[29161] = {X 295.2082, Y 93.6975, Z -2.1667, A 0.000, B 0.000, C 0.000 }
gfCNCPoint1[29162] = {X 295.9270, Y 94.3623, Z -2.1667, A 0.000, B 0.000, C 0.000 }
gfCNCPoint1[29163] = {X 296.4721, Y 95.1758, Z -2.1667, A 0.000, B 0.000, C 0.000 }
gfCNCPoint1[29164] = {X 296.8137, Y 96.0934, Z -2.1667, A 0.000, B 0.000, C 0.000 }
gfCNCPoint1[29165] = {X 296.9331, Y 97.0653, Z -2.1667, A 0.000, B 0.000, C 0.000 }
gfCNCPoint1[29166] = {X 296.9331, Y 98.0000, Z -2.1667, A 0.000, B 0.000, C 0.000 }
gfCNCPoint1[29167] = {X 296.8288, Y 98.9257, Z -2.1667, A 0.000, B 0.000, C 0.000 }
gfCNCPoint1[29168] = {X 296.5211, Y 99.8050, Z -2.1667, A 0.000, B 0.000, C 0.000 }
gfCNCPoint1[29169] = {X 296.0255, Y 100.5937, Z -2.1667, A 0.000, B 0.000, C 0.000 }
gfCNCPoint1[29170] = {X 295.3668, Y 101.2524, Z -2.1667, A 0.000, B 0.000, C 0.000 }
gfCNCPoint1[29171] = {X 294.5780, Y 101.7480, Z -2.1667, A 0.000, B 0.000, C 0.000 }
gfCNCPoint1[29172] = {X 293.6988, Y 102.0557, Z -2.1667, A 0.000, B 0.000, C 0.000 }
gfCNCPoint1[29173] = {X 292.7731, Y 102.1600, Z -2.1667, A 0.000, B 0.000, C 0.000 }
gfCNCPoint1[29174] = {X 276.2327, Y 102.1600, Z -2.1667, A 0.000, B 0.000, C 0.000 }
gfCNCPoint1[29175] = {X 275.3070, Y 102.0557, Z -2.1667, A 0.000, B 0.000, C 0.000 }
gfCNCPoint1[29176] = {X 274.4277, Y 101.7480, Z -2.1667, A 0.000, B 0.000, C 0.000 }
gfCNCPoint1[29177] = {X 273.6390, Y 101.2524, Z -2.1667, A 0.000, B 0.000, C 0.000 }
gfCNCPoint1[29178] = {X 272.9803, Y 100.5937, Z -2.1667, A 0.000, B 0.000, C 0.000 }
gfCNCPoint1[29179] = {X 272.4847, Y 99.8050, Z -2.1667, A 0.000, B 0.000, C 0.000 }
gfCNCPoint1[29180] = {X 272.1770, Y 98.9257, Z -2.1667, A 0.000, B 0.000, C 0.000 }
gfCNCPoint1[29181] = {X 272.0727, Y 98.0000, Z -2.1667, A 0.000, B 0.000, C 0.000 }
gfCNCPoint1[29182] = {X 272.0727, Y 97.0659, Z -2.1667, A 0.000, B 0.000, C 0.000 }
gfCNCPoint1[29183] = {X 272.1633, Y 96.2022, Z -2.1667, A 0.000, B 0.000, C 0.000 }
gfCNCPoint1[29184] = {X 272.4314, Y 95.3761, Z -2.1667, A 0.000, B 0.000, C 0.000 }
gfCNCPoint1[29185] = {X 272.8650, Y 94.6237, Z -2.1667, A 0.000, B 0.000, C 0.000 }
gfCNCPoint1[29186] = {X 273.4455, Y 93.9777, Z -2.1667, A 0.000, B 0.000, C 0.000 }
gfCNCPoint1[29187] = {X 274.1474, Y 93.4663, Z -2.1667, A 0.000, B 0.000, C 0.000 }
gfCNCPoint1[29188] = {X 274.9402, Y 93.1118, Z -2.1667, A 0.000, B 0.000, C 0.000 }
gfCNCPoint1[29189] = {X 275.7894, Y 92.9296, Z -2.1667, A 0.000, B 0.000, C 0.000 }
gfCNCPoint1[29190] = {X 275.7894, Y 85.4858, Z -2.1667, A 0.000, B 0.000, C 0.000 }
gfCNCPoint1[29191] = {X 262.6227, Y 80.3245, Z -2.1667, A 0.000, B 0.000, C 0.000 }
gfCNCPoint1[29192] = {X 262.1898, Y 80.5968, Z -2.1667, A 0.000, B 0.000, C 0.000 }
gfCNCPoint1[29193] = {X 237.6352, Y 96.5014, Z -2.1667, A 0.000, B 0.000, C 0.000 }
gfCNCPoint1[29194] = {X 237.6398, Y 97.0653, Z -2.1667, A 0.000, B 0.000, C 0.000 }
gfCNCPoint1[29195] = {X 237.6398, Y 98.0000, Z -2.1667, A 0.000, B 0.000, C 0.000 }
gfCNCPoint1[29196] = {X 237.5355, Y 98.9257, Z -2.1667, A 0.000, B 0.000, C 0.000 }
gfCNCPoint1[29197] = {X 237.2278, Y 99.8050, Z -2.1667, A 0.000, B 0.000, C 0.000 }
gfCNCPoint1[29198] = {X 236.7322, Y 100.5937, Z -2.1667, A 0.000, B 0.000, C 0.000 }
gfCNCPoint1[29199] = {X 236.0735, Y 101.2524, Z -2.1667, A 0.000, B 0.000, C 0.000 }
gfCNCPoint1[29200] = {X 235.2847, Y 101.7480, Z -2.1667, A 0.000, B 0.000, C 0.000 }
gfCNCPoint1[29201] = {X 234.4055, Y 102.0557, Z -2.1667, A 0.000, B 0.000, C 0.000 }
gfCNCPoint1[29202] = {X 233.4798, Y 102.1600, Z -2.1667, A 0.000, B 0.000, C 0.000 }
gfCNCPoint1[29203] = {X 214.1790, Y 102.1600, Z -2.1667, A 0.000, B 0.000, C 0.000 }
gfCNCPoint1[29204] = {X 213.7860, Y 102.1414, Z -2.1667, A 0.000, B 0.000, C 0.000 }
gfCNCPoint1[29205] = {X 213.3966, Y 102.0857, Z -2.1667, A 0.000, B 0.000, C 0.000 }
gfCNCPoint1[29206] = {X 213.0071, Y 102.1414, Z -2.1667, A 0.000, B 0.000, C 0.000 }
gfCNCPoint1[29207] = {X 212.6141, Y 102.1600, Z -2.1667, A 0.000, B 0.000, C 0.000 }
gfCNCPoint1[29208] = {X 194.9870, Y 102.1600, Z -2.1667, A 0.000, B 0.000, C 0.000 }
gfCNCPoint1[29209] = {X 194.0613, Y 102.0557, Z -2.1667, A 0.000, B 0.000, C 0.000 }
gfCNCPoint1[29210] = {X 193.1820, Y 101.7480, Z -2.1667, A 0.000, B 0.000, C 0.000 }
gfCNCPoint1[29211] = {X 192.3932, Y 101.2524, Z -2.1667, A 0.000, B 0.000, C 0.000 }
gfCNCPoint1[29212] = {X 191.7345, Y 100.5937, Z -2.1667, A 0.000, B 0.000, C 0.000 }
gfCNCPoint1[29213] = {X 191.2389, Y 99.8050, Z -2.1667, A 0.000, B 0.000, C 0.000 }
gfCNCPoint1[29214] = {X 190.9313, Y 98.9257, Z -2.1667, A 0.000, B 0.000, C 0.000 }
gfCNCPoint1[29215] = {X 190.8270, Y 98.0000, Z -2.1667, A 0.000, B 0.000, C 0.000 }
gfCNCPoint1[29216] = {X 190.8270, Y 97.0659, Z -2.1667, A 0.000, B 0.000, C 0.000 }
gfCNCPoint1[29217] = {X 190.9241, Y 96.1723, Z -2.1667, A 0.000, B 0.000, C 0.000 }
gfCNCPoint1[29218] = {X 191.2109, Y 95.3203, Z -2.1667, A 0.000, B 0.000, C 0.000 }
gfCNCPoint1[29219] = {X 191.6741, Y 94.5499, Z -2.1667, A 0.000, B 0.000, C 0.000 }
gfCNCPoint1[29220] = {X 191.7354, Y 94.4712, Z -2.1667, A 0.000, B 0.000, C 0.000 }
gfCNCPoint1[29221] = {X 191.7986, Y 94.3939, Z -2.1667, A 0.000, B 0.000, C 0.000 }
gfCNCPoint1[29222] = {X 188.6351, Y 90.9402, Z -2.1667, A 0.000, B 0.000, C 0.000 }
gfCNCPoint1[29223] = {X 150.0187, Y 90.9402, Z -2.1667, A 0.000, B 0.000, C 0.000 }
gfCNCPoint1[29224] = {X 146.9330, Y 94.3588, Z -2.1667, A 0.000, B 0.000, C 0.000 }
gfCNCPoint1[29225] = {X 147.4788, Y 95.1732, Z -2.1667, A 0.000, B 0.000, C 0.000 }
gfCNCPoint1[29226] = {X 147.8204, Y 96.0922, Z -2.1667, A 0.000, B 0.000, C 0.000 }
gfCNCPoint1[29227] = {X 147.9391, Y 97.0655, Z -2.1667, A 0.000, B 0.000, C 0.000 }
gfCNCPoint1[29228] = {X 147.9391, Y 98.0000, Z -2.1667, A 0.000, B 0.000, C 0.000 }
gfCNCPoint1[29229] = {X 147.8348, Y 98.9257, Z -2.1667, A 0.000, B 0.000, C 0.000 }
gfCNCPoint1[29230] = {X 147.5271, Y 99.8050, Z -2.1667, A 0.000, B 0.000, C 0.000 }
gfCNCPoint1[29231] = {X 147.0315, Y 100.5937, Z -2.1667, A 0.000, B 0.000, C 0.000 }
gfCNCPoint1[29232] = {X 146.3728, Y 101.2524, Z -2.1667, A 0.000, B 0.000, C 0.000 }
gfCNCPoint1[29233] = {X 145.5841, Y 101.7480, Z -2.1667, A 0.000, B 0.000, C 0.000 }
gfCNCPoint1[29234] = {X 144.7048, Y 102.0557, Z -2.1667, A 0.000, B 0.000, C 0.000 }
gfCNCPoint1[29235] = {X 143.7791, Y 102.1600, Z -2.1667, A 0.000, B 0.000, C 0.000 }
gfCNCPoint1[29236] = {X 125.0000, Y 102.1600, Z -2.1667, A 0.000, B 0.000, C 0.000 }
gfCNCPoint1[29237] = {X 124.0743, Y 102.0557, Z -2.1667, A 0.000, B 0.000, C 0.000 }
gfCNCPoint1[29238] = {X 123.1950, Y 101.7480, Z -2.1667, A 0.000, B 0.000, C 0.000 }
gfCNCPoint1[29239] = {X 122.4063, Y 101.2524, Z -2.1667, A 0.000, B 0.000, C 0.000 }
gfCNCPoint1[29240] = {X 121.7476, Y 100.5937, Z -2.1667, A 0.000, B 0.000, C 0.000 }
gfCNCPoint1[29241] = {X 121.2520, Y 99.8050, Z -2.1667, A 0.000, B 0.000, C 0.000 }
gfCNCPoint1[29242] = {X 120.9443, Y 98.9257, Z -2.1667, A 0.000, B 0.000, C 0.000 }
gfCNCPoint1[29243] = {X 120.8400, Y 98.0000, Z -2.1667, A 0.000, B 0.000, C 0.000 }
gfCNCPoint1[29244] = {X 120.8400, Y 97.0659, Z -2.1667, A 0.000, B 0.000, C 0.000 }
gfCNCPoint1[29245] = {X 120.9406, Y 96.1565, Z -2.1667, A 0.000, B 0.000, C 0.000 }
gfCNCPoint1[29246] = {X 121.2376, Y 95.2910, Z -2.1667, A 0.000, B 0.000, C 0.000 }
gfCNCPoint1[29247] = {X 121.7167, Y 94.5114, Z -2.1667, A 0.000, B 0.000, C 0.000 }
gfCNCPoint1[29248] = {X 122.3546, Y 93.8554, Z -2.1667, A 0.000, B 0.000, C 0.000 }
gfCNCPoint1[29249] = {X 123.1204, Y 93.3548, Z -2.1667, A 0.000, B 0.000, C 0.000 }
gfCNCPoint1[29250] = {X 123.9772, Y 93.0336, Z -2.1667, A 0.000, B 0.000, C 0.000 }
gfCNCPoint1[29251] = {X 124.8835, Y 92.9076, Z -2.1667, A 0.000, B 0.000, C 0.000 }
gfCNCPoint1[29252] = {X 124.9159, Y 92.8902, Z -2.1667, A 0.000, B 0.000, C 0.000 }
gfCNCPoint1[29253] = {X 124.9515, Y 92.8807, Z -2.1667, A 0.000, B 0.000, C 0.000 }
gfCNCPoint1[29254] = {X 125.4721, Y 92.8035, Z -2.1667, A 0.000, B 0.000, C 0.000 }
gfCNCPoint1[29255] = {X 126.3317, Y 92.6572, Z -2.1667, A 0.000, B 0.000, C 0.000 }
gfCNCPoint1[29256] = {X 127.1794, Y 92.4528, Z -2.1667, A 0.000, B 0.000, C 0.000 }
gfCNCPoint1[29257] = {X 128.4221, Y 91.2832, Z -2.1667, A 0.000, B 0.000, C 0.000 }
gfCNCPoint1[29258] = {X 129.5988, Y 90.0473, Z -2.1667, A 0.000, B 0.000, C 0.000 }
gfCNCPoint1[29259] = {X 140.7988, Y 77.7483, Z -2.1667, A 0.000, B 0.000, C 0.000 }
gfCNCPoint1[29260] = {X 137.8413, Y 75.0551, Z -2.1667, A 0.000, B 0.000, C 0.000 }
gfCNCPoint1[29261] = {X 140.8579, Y 77.8021, Z -2.1667, A 0.000, B 0.000, C 0.000 }
gfCNCPoint1[29262] = {X 155.9355, Y 61.2449, Z -2.1667, A 0.000, B 0.000, C 0.000 }
gfCNCPoint1[29263] = {X 155.5467, Y 60.5385, Z -2.1667, A 0.000, B 0.000, C 0.000 }
gfCNCPoint1[29264] = {X 155.3044, Y 59.7695, Z -2.1667, A 0.000, B 0.000, C 0.000 }
gfCNCPoint1[29265] = {X 155.2181, Y 58.9678, Z -2.1667, A 0.000, B 0.000, C 0.000 }
gfCNCPoint1[29266] = {X 155.2180, Y 58.0000, Z -2.1667, A 0.000, B 0.000, C 0.000 }
gfCNCPoint1[29267] = {X 155.3203, Y 57.0921, Z -2.1667, A 0.000, B 0.000, C 0.000 }
gfCNCPoint1[29268] = {X 155.6220, Y 56.2298, Z -2.1667, A 0.000, B 0.000, C 0.000 }
gfCNCPoint1[29269] = {X 156.1081, Y 55.4562, Z -2.1667, A 0.000, B 0.000, C 0.000 }
gfCNCPoint1[29270] = {X 156.7541, Y 54.8101, Z -2.1667, A 0.000, B 0.000, C 0.000 }
gfCNCPoint1[29271] = {X 157.5277, Y 54.3240, Z -2.1667, A 0.000, B 0.000, C 0.000 }
gfCNCPoint1[29272] = {X 158.3901, Y 54.0223, Z -2.1667, A 0.000, B 0.000, C 0.000 }
gfCNCPoint1[29273] = {X 159.2980, Y 53.9200, Z -2.1667, A 0.000, B 0.000, C 0.000 }
gfCNCPoint1[29274] = {X 178.5335, Y 53.9200, Z -2.1667, A 0.000, B 0.000, C 0.000 }
gfCNCPoint1[29275] = {X 179.4414, Y 54.0223, Z -2.1667, A 0.000, B 0.000, C 0.000 }
gfCNCPoint1[29276] = {X 180.3037, Y 54.3240, Z -2.1667, A 0.000, B 0.000, C 0.000 }
gfCNCPoint1[29277] = {X 181.0773, Y 54.8101, Z -2.1667, A 0.000, B 0.000, C 0.000 }
gfCNCPoint1[29278] = {X 181.7234, Y 55.4562, Z -2.1667, A 0.000, B 0.000, C 0.000 }
gfCNCPoint1[29279] = {X 182.2095, Y 56.2298, Z -2.1667, A 0.000, B 0.000, C 0.000 }
gfCNCPoint1[29280] = {X 182.5112, Y 57.0921, Z -2.1667, A 0.000, B 0.000, C 0.000 }
gfCNCPoint1[29281] = {X 182.6135, Y 58.0000, Z -2.1667, A 0.000, B 0.000, C 0.000 }
gfCNCPoint1[29282] = {X 182.6135, Y 58.9342, Z -2.1667, A 0.000, B 0.000, C 0.000 }
gfCNCPoint1[29283] = {X 182.5334, Y 59.7386, Z -2.1667, A 0.000, B 0.000, C 0.000 }
gfCNCPoint1[29284] = {X 182.2963, Y 60.5114, Z -2.1667, A 0.000, B 0.000, C 0.000 }
gfCNCPoint1[29285] = {X 181.9114, Y 61.2223, Z -2.1667, A 0.000, B 0.000, C 0.000 }
gfCNCPoint1[29286] = {X 209.3006, Y 91.1160, Z -2.1667, A 0.000, B 0.000, C 0.000 }
gfCNCPoint1[29287] = {X 209.9710, Y 91.7962, Z -2.1667, A 0.000, B 0.000, C 0.000 }
gfCNCPoint1[29288] = {X 210.6891, Y 92.4257, Z -2.1667, A 0.000, B 0.000, C 0.000 }
gfCNCPoint1[29289] = {X 211.0139, Y 92.6307, Z -2.1667, A 0.000, B 0.000, C 0.000 }
gfCNCPoint1[29290] = {X 211.3781, Y 92.7524, Z -2.1667, A 0.000, B 0.000, C 0.000 }
gfCNCPoint1[29291] = {X 213.3970, Y 93.0674, Z -2.1667, A 0.000, B 0.000, C 0.000 }
gfCNCPoint1[29292] = {X 214.4547, Y 92.9774, Z -2.1667, A 0.000, B 0.000, C 0.000 }
gfCNCPoint1[29293] = {X 215.5145, Y 92.9165, Z -2.1667, A 0.000, B 0.000, C 0.000 }
gfCNCPoint1[29294] = {X 216.2276, Y 92.8378, Z -2.1667, A 0.000, B 0.000, C 0.000 }
gfCNCPoint1[29295] = {X 216.9142, Y 92.6299, Z -2.1667, A 0.000, B 0.000, C 0.000 }
gfCNCPoint1[29296] = {X 217.5511, Y 92.2998, Z -2.1667, A 0.000, B 0.000, C 0.000 }
gfCNCPoint1[29297] = {X 223.0910, Y 88.7245, Z -2.1667, A 0.000, B 0.000, C 0.000 }
gfCNCPoint1[29298] = {X 246.3550, Y 73.8480, Z -2.1667, A 0.000, B 0.000, C 0.000 }
gfCNCPoint1[29299] = {X 221.7196, Y 64.1799, Z -2.1667, A 0.000, B 0.000, C 0.000 }
gfCNCPoint1[29300] = {X 219.9262, Y 63.5796, Z -2.1667, A 0.000, B 0.000, C 0.000 }
gfCNCPoint1[29301] = {X 218.0758, Y 63.1885, Z -2.1667, A 0.000, B 0.000, C 0.000 }
gfCNCPoint1[29302] = {X 216.1929, Y 63.0117, Z -2.1667, A 0.000, B 0.000, C 0.000 }
gfCNCPoint1[29303] = {X 215.3127, Y 62.8850, Z -2.1667, A 0.000, B 0.000, C 0.000 }
gfCNCPoint1[29304] = {X 214.4809, Y 62.5706, Z -2.1667, A 0.000, B 0.000, C 0.000 }
gfCNCPoint1[29305] = {X 213.7370, Y 62.0834, Z -2.1667, A 0.000, B 0.000, C 0.000 }
gfCNCPoint1[29306] = {X 213.1162, Y 61.4466, Z -2.1667, A 0.000, B 0.000, C 0.000 }
gfCNCPoint1[29307] = {X 212.6482, Y 60.6905, Z -2.1667, A 0.000, B 0.000, C 0.000 }
gfCNCPoint1[29308] = {X 212.3552, Y 59.8509, Z -2.1667, A 0.000, B 0.000, C 0.000 }
gfCNCPoint1[29309] = {X 212.2509, Y 58.9678, Z -2.1667, A 0.000, B 0.000, C 0.000 }
gfCNCPoint1[29310] = {X 212.2508, Y 58.0000, Z -2.1667, A 0.000, B 0.000, C 0.000 }
gfCNCPoint1[29311] = {X 212.3531, Y 57.0921, Z -2.1667, A 0.000, B 0.000, C 0.000 }
gfCNCPoint1[29312] = {X 212.6549, Y 56.2298, Z -2.1667, A 0.000, B 0.000, C 0.000 }
gfCNCPoint1[29313] = {X 213.1409, Y 55.4562, Z -2.1667, A 0.000, B 0.000, C 0.000 }
gfCNCPoint1[29314] = {X 213.7870, Y 54.8101, Z -2.1667, A 0.000, B 0.000, C 0.000 }
gfCNCPoint1[29315] = {X 214.5606, Y 54.3240, Z -2.1667, A 0.000, B 0.000, C 0.000 }
gfCNCPoint1[29316] = {X 215.4229, Y 54.0223, Z -2.1667, A 0.000, B 0.000, C 0.000 }
gfCNCPoint1[29317] = {X 216.3308, Y 53.9200, Z -2.1667, A 0.000, B 0.000, C 0.000 }
gfCNCPoint1[29318] = {X 237.2617, Y 53.9200, Z -2.1667, A 0.000, B 0.000, C 0.000 }
gfCNCPoint1[29319] = {X 238.1696, Y 54.0223, Z -2.1667, A 0.000, B 0.000, C 0.000 }
gfCNCPoint1[29320] = {X 239.0319, Y 54.3240, Z -2.1667, A 0.000, B 0.000, C 0.000 }
gfCNCPoint1[29321] = {X 239.8055, Y 54.8101, Z -2.1667, A 0.000, B 0.000, C 0.000 }
gfCNCPoint1[29322] = {X 240.4516, Y 55.4562, Z -2.1667, A 0.000, B 0.000, C 0.000 }
gfCNCPoint1[29323] = {X 240.9376, Y 56.2298, Z -2.1667, A 0.000, B 0.000, C 0.000 }
gfCNCPoint1[29324] = {X 241.2394, Y 57.0921, Z -2.1667, A 0.000, B 0.000, C 0.000 }
gfCNCPoint1[29325] = {X 241.3417, Y 58.0000, Z -2.1667, A 0.000, B 0.000, C 0.000 }
gfCNCPoint1[29326] = {X 241.3417, Y 58.3969, Z -2.1667, A 0.000, B 0.000, C 0.000 }
gfCNCPoint1[29327] = {X 247.4005, Y 60.7590, Z -2.1667, A 0.000, B 0.000, C 0.000 }
gfCNCPoint1[29328] = {X 275.8738, Y 72.0564, Z -2.1667, A 0.000, B 0.000, C 0.000 }
gfCNCPoint1[29329] = {X 275.8745, Y 62.9983, Z -2.1667, A 0.000, B 0.000, C 0.000 }
gfCNCPoint1[29330] = {X 275.7382, Y 62.9840, Z -2.1667, A 0.000, B 0.000, C 0.000 }
gfCNCPoint1[29331] = {X 275.6025, Y 62.9651, Z -2.1667, A 0.000, B 0.000, C 0.000 }
gfCNCPoint1[29332] = {X 274.6828, Y 62.7082, Z -2.1667, A 0.000, B 0.000, C 0.000 }
gfCNCPoint1[29333] = {X 273.8480, Y 62.2446, Z -2.1667, A 0.000, B 0.000, C 0.000 }
gfCNCPoint1[29334] = {X 273.1439, Y 61.5997, Z -2.1667, A 0.000, B 0.000, C 0.000 }
gfCNCPoint1[29335] = {X 272.6089, Y 60.8087, Z -2.1667, A 0.000, B 0.000, C 0.000 }
gfCNCPoint1[29336] = {X 272.2724, Y 59.9151, Z -2.1667, A 0.000, B 0.000, C 0.000 }
gfCNCPoint1[29337] = {X 272.1528, Y 58.9678, Z -2.1667, A 0.000, B 0.000, C 0.000 }
gfCNCPoint1[29338] = {X 272.1527, Y 58.0000, Z -2.1667, A 0.000, B 0.000, C 0.000 }
gfCNCPoint1[29339] = {X 272.2550, Y 57.0921, Z -2.1667, A 0.000, B 0.000, C 0.000 }
gfCNCPoint1[29340] = {X 272.5567, Y 56.2298, Z -2.1667, A 0.000, B 0.000, C 0.000 }
gfCNCPoint1[29341] = {X 273.0428, Y 55.4562, Z -2.1667, A 0.000, B 0.000, C 0.000 }
gfCNCPoint1[29342] = {X 273.6889, Y 54.8101, Z -2.1667, A 0.000, B 0.000, C 0.000 }
gfCNCPoint1[29343] = {X 274.4624, Y 54.3240, Z -2.1667, A 0.000, B 0.000, C 0.000 }
gfCNCPoint1[29344] = {X 275.3248, Y 54.0223, Z -2.1667, A 0.000, B 0.000, C 0.000 }
gfCNCPoint1[29345] = {X 276.2327, Y 53.9200, Z -2.1667, A 0.000, B 0.000, C 0.000 }
gfCNCPoint1[29346] = {X 292.7731, Y 53.9200, Z -2.1667, A 0.000, B 0.000, C 0.000 }
gfCNCPoint1[29347] = {X 293.6810, Y 54.0223, Z -2.1667, A 0.000, B 0.000, C 0.000 }
gfCNCPoint1[29348] = {X 294.5433, Y 54.3240, Z -2.1667, A 0.000, B 0.000, C 0.000 }
gfCNCPoint1[29349] = {X 295.3169, Y 54.8101, Z -2.1667, A 0.000, B 0.000, C 0.000 }
gfCNCPoint1[29350] = {X 295.9630, Y 55.4562, Z -2.1667, A 0.000, B 0.000, C 0.000 }
gfCNCPoint1[29351] = {X 296.4490, Y 56.2298, Z -2.1667, A 0.000, B 0.000, C 0.000 }
gfCNCPoint1[29352] = {X 296.7508, Y 57.0921, Z -2.1667, A 0.000, B 0.000, C 0.000 }
gfCNCPoint1[29353] = {X 296.8531, Y 58.0000, Z -2.1667, A 0.000, B 0.000, C 0.000 }
gfCNCPoint1[29354] = {X 296.8531, Y 58.9344, Z -2.1667, A 0.000, B 0.000, C 0.000 }
gfCNCPoint1[29355] = {X 296.7373, Y 59.8874, Z -2.1667, A 0.000, B 0.000, C 0.000 }
gfCNCPoint1[29356] = {X 296.4029, Y 60.7873, Z -2.1667, A 0.000, B 0.000, C 0.000 }
gfCNCPoint1[29357] = {X 295.8683, Y 61.5847, Z -2.1667, A 0.000, B 0.000, C 0.000 }
gfCNCPoint1[29358] = {X 295.1628, Y 62.2358, Z -2.1667, A 0.000, B 0.000, C 0.000 }
gfCNCPoint1[29359] = {X 294.3252, Y 62.7048, Z -2.1667, A 0.000, B 0.000, C 0.000 }
gfCNCPoint1[29360] = {X 293.4014, Y 62.9660, Z -2.1667, A 0.000, B 0.000, C 0.000 }
gfCNCPoint1[29361] = {X 293.2750, Y 62.9841, Z -2.1667, A 0.000, B 0.000, C 0.000 }
gfCNCPoint1[29362] = {X 293.1480, Y 62.9983, Z -2.1667, A 0.000, B 0.000, C 0.000 }
gfCNCPoint1[29363] = {X 293.1318, Y 63.1581, Z -2.1667, A 0.000, B 0.000, C 0.000 }
gfCNCPoint1[29364] = {X 293.1442, Y 92.9941, Z -2.1667, A 0.000, B 0.000, C 0.000 }
gfCNCPoint1[29365] = {X 293.2726, Y 93.0088, Z -2.1667, A 0.000, B 0.000, C 0.000 }
gfCNCPoint1[29366] = {X 293.4004, Y 93.0275, Z -2.1667, A 0.000, B 0.000, C 0.000 }
gfCNCPoint1[29367] = {X 294.3239, Y 93.2914, Z -2.1667, A 0.000, B 0.000, C 0.000 }
gfCNCPoint1[29368] = {X 295.1611, Y 93.7622, Z -2.1667, A 0.000, B 0.000, C 0.000 }
gfCNCPoint1[29369] = {X 295.8662, Y 94.4143, Z -2.1667, A 0.000, B 0.000, C 0.000 }
gfCNCPoint1[29370] = {X 296.4009, Y 95.2122, Z -2.1667, A 0.000, B 0.000, C 0.000 }
gfCNCPoint1[29371] = {X 296.7359, Y 96.1124, Z -2.1667, A 0.000, B 0.000, C 0.000 }
gfCNCPoint1[29372] = {X 296.8531, Y 97.0657, Z -2.1667, A 0.000, B 0.000, C 0.000 }
gfCNCPoint1[29373] = {X 296.8531, Y 98.0000, Z -2.1667, A 0.000, B 0.000, C 0.000 }
gfCNCPoint1[29374] = {X 296.7508, Y 98.9079, Z -2.1667, A 0.000, B 0.000, C 0.000 }
gfCNCPoint1[29375] = {X 296.4490, Y 99.7702, Z -2.1667, A 0.000, B 0.000, C 0.000 }
gfCNCPoint1[29376] = {X 295.9630, Y 100.5438, Z -2.1667, A 0.000, B 0.000, C 0.000 }
gfCNCPoint1[29377] = {X 295.3169, Y 101.1899, Z -2.1667, A 0.000, B 0.000, C 0.000 }
gfCNCPoint1[29378] = {X 294.5433, Y 101.6760, Z -2.1667, A 0.000, B 0.000, C 0.000 }
gfCNCPoint1[29379] = {X 293.6810, Y 101.9777, Z -2.1667, A 0.000, B 0.000, C 0.000 }
gfCNCPoint1[29380] = {X 292.7731, Y 102.0800, Z -2.1667, A 0.000, B 0.000, C 0.000 }
gfCNCPoint1[29381] = {X 276.2327, Y 102.0800, Z -2.1667, A 0.000, B 0.000, C 0.000 }
gfCNCPoint1[29382] = {X 275.3248, Y 101.9777, Z -2.1667, A 0.000, B 0.000, C 0.000 }
gfCNCPoint1[29383] = {X 274.4624, Y 101.6760, Z -2.1667, A 0.000, B 0.000, C 0.000 }
gfCNCPoint1[29384] = {X 273.6889, Y 101.1899, Z -2.1667, A 0.000, B 0.000, C 0.000 }
gfCNCPoint1[29385] = {X 273.0428, Y 100.5438, Z -2.1667, A 0.000, B 0.000, C 0.000 }
gfCNCPoint1[29386] = {X 272.5567, Y 99.7702, Z -2.1667, A 0.000, B 0.000, C 0.000 }
gfCNCPoint1[29387] = {X 272.2550, Y 98.9079, Z -2.1667, A 0.000, B 0.000, C 0.000 }
gfCNCPoint1[29388] = {X 272.1527, Y 98.0000, Z -2.1667, A 0.000, B 0.000, C 0.000 }
gfCNCPoint1[29389] = {X 272.1527, Y 97.0659, Z -2.1667, A 0.000, B 0.000, C 0.000 }
gfCNCPoint1[29390] = {X 272.2437, Y 96.2088, Z -2.1667, A 0.000, B 0.000, C 0.000 }
gfCNCPoint1[29391] = {X 272.5128, Y 95.3899, Z -2.1667, A 0.000, B 0.000, C 0.000 }
gfCNCPoint1[29392] = {X 272.9480, Y 94.6458, Z -2.1667, A 0.000, B 0.000, C 0.000 }
gfCNCPoint1[29393] = {X 273.5297, Y 94.0098, Z -2.1667, A 0.000, B 0.000, C 0.000 }
gfCNCPoint1[29394] = {X 274.2321, Y 93.5101, Z -2.1667, A 0.000, B 0.000, C 0.000 }
gfCNCPoint1[29395] = {X 275.0238, Y 93.1692, Z -2.1667, A 0.000, B 0.000, C 0.000 }
gfCNCPoint1[29396] = {X 275.8694, Y 93.0021, Z -2.1667, A 0.000, B 0.000, C 0.000 }
gfCNCPoint1[29397] = {X 275.8694, Y 85.4313, Z -2.1667, A 0.000, B 0.000, C 0.000 }
gfCNCPoint1[29398] = {X 262.6143, Y 80.2352, Z -2.1667, A 0.000, B 0.000, C 0.000 }
gfCNCPoint1[29399] = {X 262.1467, Y 80.5294, Z -2.1667, A 0.000, B 0.000, C 0.000 }
gfCNCPoint1[29400] = {X 237.5549, Y 96.4581, Z -2.1667, A 0.000, B 0.000, C 0.000 }
gfCNCPoint1[29401] = {X 237.5598, Y 97.0656, Z -2.1667, A 0.000, B 0.000, C 0.000 }
gfCNCPoint1[29402] = {X 237.5598, Y 98.0000, Z -2.1667, A 0.000, B 0.000, C 0.000 }
gfCNCPoint1[29403] = {X 237.4575, Y 98.9079, Z -2.1667, A 0.000, B 0.000, C 0.000 }
gfCNCPoint1[29404] = {X 237.1557, Y 99.7702, Z -2.1667, A 0.000, B 0.000, C 0.000 }
gfCNCPoint1[29405] = {X 236.6697, Y 100.5438, Z -2.1667, A 0.000, B 0.000, C 0.000 }
gfCNCPoint1[29406] = {X 236.0236, Y 101.1899, Z -2.1667, A 0.000, B 0.000, C 0.000 }
gfCNCPoint1[29407] = {X 235.2500, Y 101.6760, Z -2.1667, A 0.000, B 0.000, C 0.000 }
gfCNCPoint1[29408] = {X 234.3877, Y 101.9777, Z -2.1667, A 0.000, B 0.000, C 0.000 }
gfCNCPoint1[29409] = {X 233.4798, Y 102.0800, Z -2.1667, A 0.000, B 0.000, C 0.000 }
gfCNCPoint1[29410] = {X 214.1790, Y 102.0800, Z -2.1667, A 0.000, B 0.000, C 0.000 }
gfCNCPoint1[29411] = {X 213.7860, Y 102.0610, Z -2.1667, A 0.000, B 0.000, C 0.000 }
gfCNCPoint1[29412] = {X 213.3966, Y 102.0043, Z -2.1667, A 0.000, B 0.000, C 0.000 }
gfCNCPoint1[29413] = {X 213.0072, Y 102.0610, Z -2.1667, A 0.000, B 0.000, C 0.000 }
gfCNCPoint1[29414] = {X 212.6141, Y 102.0800, Z -2.1667, A 0.000, B 0.000, C 0.000 }
gfCNCPoint1[29415] = {X 194.9870, Y 102.0800, Z -2.1667, A 0.000, B 0.000, C 0.000 }
gfCNCPoint1[29416] = {X 194.0791, Y 101.9777, Z -2.1667, A 0.000, B 0.000, C 0.000 }
gfCNCPoint1[29417] = {X 193.2167, Y 101.6760, Z -2.1667, A 0.000, B 0.000, C 0.000 }
gfCNCPoint1[29418] = {X 192.4431, Y 101.1899, Z -2.1667, A 0.000, B 0.000, C 0.000 }
gfCNCPoint1[29419] = {X 191.7971, Y 100.5438, Z -2.1667, A 0.000, B 0.000, C 0.000 }
gfCNCPoint1[29420] = {X 191.3110, Y 99.7702, Z -2.1667, A 0.000, B 0.000, C 0.000 }
gfCNCPoint1[29421] = {X 191.0093, Y 98.9079, Z -2.1667, A 0.000, B 0.000, C 0.000 }
gfCNCPoint1[29422] = {X 190.9070, Y 98.0000, Z -2.1667, A 0.000, B 0.000, C 0.000 }
gfCNCPoint1[29423] = {X 190.9070, Y 97.0659, Z -2.1667, A 0.000, B 0.000, C 0.000 }
gfCNCPoint1[29424] = {X 191.0022, Y 96.1894, Z -2.1667, A 0.000, B 0.000, C 0.000 }
gfCNCPoint1[29425] = {X 191.2835, Y 95.3539, Z -2.1667, A 0.000, B 0.000, C 0.000 }
gfCNCPoint1[29426] = {X 191.7378, Y 94.5983, Z -2.1667, A 0.000, B 0.000, C 0.000 }
gfCNCPoint1[29427] = {X 191.8199, Y 94.4938, Z -2.1667, A 0.000, B 0.000, C 0.000 }
gfCNCPoint1[29428] = {X 191.9053, Y 94.3920, Z -2.1667, A 0.000, B 0.000, C 0.000 }
gfCNCPoint1[29429] = {X 188.6703, Y 90.8602, Z -2.1667, A 0.000, B 0.000, C 0.000 }
gfCNCPoint1[29430] = {X 149.9831, Y 90.8602, Z -2.1667, A 0.000, B 0.000, C 0.000 }
gfCNCPoint1[29431] = {X 146.8261, Y 94.3578, Z -2.1667, A 0.000, B 0.000, C 0.000 }
gfCNCPoint1[29432] = {X 147.3860, Y 95.1682, Z -2.1667, A 0.000, B 0.000, C 0.000 }
gfCNCPoint1[29433] = {X 147.7371, Y 96.0884, Z -2.1667, A 0.000, B 0.000, C 0.000 }
gfCNCPoint1[29434] = {X 147.8591, Y 97.0658, Z -2.1667, A 0.000, B 0.000, C 0.000 }
gfCNCPoint1[29435] = {X 147.8591, Y 98.0000, Z -2.1667, A 0.000, B 0.000, C 0.000 }
gfCNCPoint1[29436] = {X 147.7568, Y 98.9079, Z -2.1667, A 0.000, B 0.000, C 0.000 }
gfCNCPoint1[29437] = {X 147.4551, Y 99.7702, Z -2.1667, A 0.000, B 0.000, C 0.000 }
gfCNCPoint1[29438] = {X 146.9690, Y 100.5438, Z -2.1667, A 0.000, B 0.000, C 0.000 }
gfCNCPoint1[29439] = {X 146.3229, Y 101.1899, Z -2.1667, A 0.000, B 0.000, C 0.000 }
gfCNCPoint1[29440] = {X 145.5494, Y 101.6760, Z -2.1667, A 0.000, B 0.000, C 0.000 }
gfCNCPoint1[29441] = {X 144.6870, Y 101.9777, Z -2.1667, A 0.000, B 0.000, C 0.000 }
gfCNCPoint1[29442] = {X 143.7791, Y 102.0800, Z -2.1667, A 0.000, B 0.000, C 0.000 }
gfCNCPoint1[29443] = {X 125.0000, Y 102.0800, Z -2.1667, A 0.000, B 0.000, C 0.000 }
gfCNCPoint1[29444] = {X 124.0921, Y 101.9777, Z -2.1667, A 0.000, B 0.000, C 0.000 }
gfCNCPoint1[29445] = {X 123.2298, Y 101.6760, Z -2.1667, A 0.000, B 0.000, C 0.000 }
gfCNCPoint1[29446] = {X 122.4562, Y 101.1899, Z -2.1667, A 0.000, B 0.000, C 0.000 }
gfCNCPoint1[29447] = {X 121.8101, Y 100.5438, Z -2.1667, A 0.000, B 0.000, C 0.000 }
gfCNCPoint1[29448] = {X 121.3240, Y 99.7702, Z -2.1667, A 0.000, B 0.000, C 0.000 }
gfCNCPoint1[29449] = {X 121.0223, Y 98.9079, Z -2.1667, A 0.000, B 0.000, C 0.000 }
gfCNCPoint1[29450] = {X 120.9200, Y 98.0000, Z -2.1667, A 0.000, B 0.000, C 0.000 }
gfCNCPoint1[29451] = {X 120.9200, Y 97.0659, Z -2.1667, A 0.000, B 0.000, C 0.000 }
gfCNCPoint1[29452] = {X 121.0194, Y 96.1709, Z -2.1667, A 0.000, B 0.000, C 0.000 }
gfCNCPoint1[29453] = {X 121.3127, Y 95.3194, Z -2.1667, A 0.000, B 0.000, C 0.000 }
gfCNCPoint1[29454] = {X 121.7857, Y 94.5531, Z -2.1667, A 0.000, B 0.000, C 0.000 }
gfCNCPoint1[29455] = {X 122.4152, Y 93.9091, Z -2.1667, A 0.000, B 0.000, C 0.000 }
gfCNCPoint1[29456] = {X 123.1707, Y 93.4190, Z -2.1667, A 0.000, B 0.000, C 0.000 }
gfCNCPoint1[29457] = {X 124.0153, Y 93.1065, Z -2.1667, A 0.000, B 0.000, C 0.000 }
gfCNCPoint1[29458] = {X 124.9079, Y 92.9870, Z -2.1667, A 0.000, B 0.000, C 0.000 }
gfCNCPoint1[29459] = {X 124.9317, Y 92.9717, Z -2.1667, A 0.000, B 0.000, C 0.000 }
gfCNCPoint1[29460] = {X 124.9632, Y 92.9599, Z -2.1667, A 0.000, B 0.000, C 0.000 }
gfCNCPoint1[29461] = {X 125.4828, Y 92.8828, Z -2.1667, A 0.000, B 0.000, C 0.000 }
gfCNCPoint1[29462] = {X 126.3569, Y 92.7337, Z -2.1667, A 0.000, B 0.000, C 0.000 }
gfCNCPoint1[29463] = {X 127.2187, Y 92.5249, Z -2.1667, A 0.000, B 0.000, C 0.000 }
gfCNCPoint1[29464] = {X 128.4719, Y 91.3465, Z -2.1667, A 0.000, B 0.000, C 0.000 }
gfCNCPoint1[29465] = {X 129.6582, Y 90.1009, Z -2.1667, A 0.000, B 0.000, C 0.000 }
gfCNCPoint1[29466] = {X 140.8579, Y 77.8021, Z -2.1667, A 0.000, B 0.000, C 0.000 }
gfCNCPoint1[29467] = {X 137.8978, Y 75.1065, Z -2.1667, A 0.000, B 0.000, C 0.000 }
gfCNCPoint1[29468] = {X 137.8982, Y 75.1061, Z -2.1667, A 0.000, B 0.000, C 0.000 }
gfCNCPoint1[29469] = {X 140.9144, Y 77.8536, Z -2.1667, A 0.000, B 0.000, C 0.000 }
gfCNCPoint1[29470] = {X 156.0377, Y 61.2515, Z -2.1667, A 0.000, B 0.000, C 0.000 }
gfCNCPoint1[29471] = {X 155.6326, Y 60.5357, Z -2.1667, A 0.000, B 0.000, C 0.000 }
gfCNCPoint1[29472] = {X 155.3825, Y 59.7522, Z -2.1667, A 0.000, B 0.000, C 0.000 }
gfCNCPoint1[29473] = {X 155.2980, Y 58.9340, Z -2.1667, A 0.000, B 0.000, C 0.000 }
gfCNCPoint1[29474] = {X 155.2980, Y 58.0000, Z -2.1667, A 0.000, B 0.000, C 0.000 }
gfCNCPoint1[29475] = {X 155.3982, Y 57.1099, Z -2.1667, A 0.000, B 0.000, C 0.000 }
gfCNCPoint1[29476] = {X 155.6941, Y 56.2645, Z -2.1667, A 0.000, B 0.000, C 0.000 }
gfCNCPoint1[29477] = {X 156.1706, Y 55.5060, Z -2.1667, A 0.000, B 0.000, C 0.000 }
gfCNCPoint1[29478] = {X 156.8040, Y 54.8727, Z -2.1667, A 0.000, B 0.000, C 0.000 }
gfCNCPoint1[29479] = {X 157.5624, Y 54.3961, Z -2.1667, A 0.000, B 0.000, C 0.000 }
gfCNCPoint1[29480] = {X 158.4079, Y 54.1003, Z -2.1667, A 0.000, B 0.000, C 0.000 }
gfCNCPoint1[29481] = {X 159.2980, Y 54.0000, Z -2.1667, A 0.000, B 0.000, C 0.000 }
gfCNCPoint1[29482] = {X 178.5335, Y 54.0000, Z -2.1667, A 0.000, B 0.000, C 0.000 }
gfCNCPoint1[29483] = {X 179.4236, Y 54.1003, Z -2.1667, A 0.000, B 0.000, C 0.000 }
gfCNCPoint1[29484] = {X 180.2690, Y 54.3961, Z -2.1667, A 0.000, B 0.000, C 0.000 }
gfCNCPoint1[29485] = {X 181.0275, Y 54.8727, Z -2.1667, A 0.000, B 0.000, C 0.000 }
gfCNCPoint1[29486] = {X 181.6608, Y 55.5060, Z -2.1667, A 0.000, B 0.000, C 0.000 }
gfCNCPoint1[29487] = {X 182.1374, Y 56.2645, Z -2.1667, A 0.000, B 0.000, C 0.000 }
gfCNCPoint1[29488] = {X 182.4332, Y 57.1099, Z -2.1667, A 0.000, B 0.000, C 0.000 }
gfCNCPoint1[29489] = {X 182.5335, Y 58.0000, Z -2.1667, A 0.000, B 0.000, C 0.000 }
gfCNCPoint1[29490] = {X 182.5334, Y 58.9671, Z -2.1667, A 0.000, B 0.000, C 0.000 }
gfCNCPoint1[29491] = {X 182.4463, Y 59.7649, Z -2.1667, A 0.000, B 0.000, C 0.000 }
gfCNCPoint1[29492] = {X 182.2017, Y 60.5293, Z -2.1667, A 0.000, B 0.000, C 0.000 }
gfCNCPoint1[29493] = {X 181.8094, Y 61.2294, Z -2.1667, A 0.000, B 0.000, C 0.000 }
gfCNCPoint1[29494] = {X 209.2416, Y 91.1700, Z -2.1667, A 0.000, B 0.000, C 0.000 }
gfCNCPoint1[29495] = {X 209.9161, Y 91.8544, Z -2.1667, A 0.000, B 0.000, C 0.000 }
gfCNCPoint1[29496] = {X 210.6386, Y 92.4878, Z -2.1667, A 0.000, B 0.000, C 0.000 }
gfCNCPoint1[29497] = {X 210.9796, Y 92.7030, Z -2.1667, A 0.000, B 0.000, C 0.000 }
gfCNCPoint1[29498] = {X 211.3621, Y 92.8308, Z -2.1667, A 0.000, B 0.000, C 0.000 }
gfCNCPoint1[29499] = {X 212.0545, Y 92.9789, Z -2.1667, A 0.000, B 0.000, C 0.000 }
gfCNCPoint1[29500] = {X 213.3959, Y 93.1479, Z -2.1667, A 0.000, B 0.000, C 0.000 }
gfCNCPoint1[29501] = {X 214.4554, Y 93.0575, Z -2.1667, A 0.000, B 0.000, C 0.000 }
gfCNCPoint1[29502] = {X 215.5170, Y 92.9965, Z -2.1667, A 0.000, B 0.000, C 0.000 }
gfCNCPoint1[29503] = {X 216.2443, Y 92.9160, Z -2.1667, A 0.000, B 0.000, C 0.000 }
gfCNCPoint1[29504] = {X 216.9447, Y 92.7038, Z -2.1667, A 0.000, B 0.000, C 0.000 }
gfCNCPoint1[29505] = {X 217.5944, Y 92.3670, Z -2.1667, A 0.000, B 0.000, C 0.000 }
gfCNCPoint1[29506] = {X 223.1343, Y 88.7918, Z -2.1667, A 0.000, B 0.000, C 0.000 }
gfCNCPoint1[29507] = {X 246.5303, Y 73.8309, Z -2.1667, A 0.000, B 0.000, C 0.000 }
gfCNCPoint1[29508] = {X 221.7493, Y 64.1056, Z -2.1667, A 0.000, B 0.000, C 0.000 }
gfCNCPoint1[29509] = {X 219.9472, Y 63.5024, Z -2.1667, A 0.000, B 0.000, C 0.000 }
gfCNCPoint1[29510] = {X 218.0879, Y 63.1094, Z -2.1667, A 0.000, B 0.000, C 0.000 }
gfCNCPoint1[29511] = {X 216.1958, Y 62.9318, Z -2.1667, A 0.000, B 0.000, C 0.000 }
gfCNCPoint1[29512] = {X 215.3283, Y 62.8064, Z -2.1667, A 0.000, B 0.000, C 0.000 }
gfCNCPoint1[29513] = {X 214.5089, Y 62.4950, Z -2.1667, A 0.000, B 0.000, C 0.000 }
gfCNCPoint1[29514] = {X 213.7770, Y 62.0127, Z -2.1667, A 0.000, B 0.000, C 0.000 }
gfCNCPoint1[29515] = {X 213.1677, Y 61.3825, Z -2.1667, A 0.000, B 0.000, C 0.000 }
gfCNCPoint1[29516] = {X 212.7104, Y 60.6348, Z -2.1667, A 0.000, B 0.000, C 0.000 }
gfCNCPoint1[29517] = {X 212.4268, Y 59.8053, Z -2.1667, A 0.000, B 0.000, C 0.000 }
gfCNCPoint1[29518] = {X 212.3308, Y 58.9340, Z -2.1667, A 0.000, B 0.000, C 0.000 }
gfCNCPoint1[29519] = {X 212.3308, Y 58.0000, Z -2.1667, A 0.000, B 0.000, C 0.000 }
gfCNCPoint1[29520] = {X 212.4311, Y 57.1099, Z -2.1667, A 0.000, B 0.000, C 0.000 }
gfCNCPoint1[29521] = {X 212.7269, Y 56.2645, Z -2.1667, A 0.000, B 0.000, C 0.000 }
gfCNCPoint1[29522] = {X 213.2035, Y 55.5060, Z -2.1667, A 0.000, B 0.000, C 0.000 }
gfCNCPoint1[29523] = {X 213.8368, Y 54.8727, Z -2.1667, A 0.000, B 0.000, C 0.000 }
gfCNCPoint1[29524] = {X 214.5953, Y 54.3961, Z -2.1667, A 0.000, B 0.000, C 0.000 }
gfCNCPoint1[29525] = {X 215.4407, Y 54.1003, Z -2.1667, A 0.000, B 0.000, C 0.000 }
gfCNCPoint1[29526] = {X 216.3308, Y 54.0000, Z -2.1667, A 0.000, B 0.000, C 0.000 }
gfCNCPoint1[29527] = {X 237.2617, Y 54.0000, Z -2.1667, A 0.000, B 0.000, C 0.000 }
gfCNCPoint1[29528] = {X 238.1518, Y 54.1003, Z -2.1667, A 0.000, B 0.000, C 0.000 }
gfCNCPoint1[29529] = {X 238.9972, Y 54.3961, Z -2.1667, A 0.000, B 0.000, C 0.000 }
gfCNCPoint1[29530] = {X 239.7556, Y 54.8727, Z -2.1667, A 0.000, B 0.000, C 0.000 }
gfCNCPoint1[29531] = {X 240.3890, Y 55.5060, Z -2.1667, A 0.000, B 0.000, C 0.000 }
gfCNCPoint1[29532] = {X 240.8656, Y 56.2645, Z -2.1667, A 0.000, B 0.000, C 0.000 }
gfCNCPoint1[29533] = {X 241.1614, Y 57.1099, Z -2.1667, A 0.000, B 0.000, C 0.000 }
gfCNCPoint1[29534] = {X 241.2617, Y 58.0000, Z -2.1667, A 0.000, B 0.000, C 0.000 }
gfCNCPoint1[29535] = {X 241.2617, Y 58.4516, Z -2.1667, A 0.000, B 0.000, C 0.000 }
gfCNCPoint1[29536] = {X 247.3712, Y 60.8334, Z -2.1667, A 0.000, B 0.000, C 0.000 }
gfCNCPoint1[29537] = {X 275.9538, Y 72.1742, Z -2.1667, A 0.000, B 0.000, C 0.000 }
gfCNCPoint1[29538] = {X 275.9530, Y 63.0380, Z -2.1667, A 0.000, B 0.000, C 0.000 }
gfCNCPoint1[29539] = {X 275.9573, Y 62.9246, Z -2.1667, A 0.000, B 0.000, C 0.000 }
gfCNCPoint1[29540] = {X 275.7857, Y 62.9090, Z -2.1667, A 0.000, B 0.000, C 0.000 }
gfCNCPoint1[29541] = {X 275.6148, Y 62.8861, Z -2.1667, A 0.000, B 0.000, C 0.000 }
gfCNCPoint1[29542] = {X 274.7081, Y 62.6321, Z -2.1667, A 0.000, B 0.000, C 0.000 }
gfCNCPoint1[29543] = {X 273.8858, Y 62.1733, Z -2.1667, A 0.000, B 0.000, C 0.000 }
gfCNCPoint1[29544] = {X 273.1936, Y 61.5349, Z -2.1667, A 0.000, B 0.000, C 0.000 }
gfCNCPoint1[29545] = {X 272.6699, Y 60.7524, Z -2.1667, A 0.000, B 0.000, C 0.000 }
gfCNCPoint1[29546] = {X 272.3435, Y 59.8691, Z -2.1667, A 0.000, B 0.000, C 0.000 }
gfCNCPoint1[29547] = {X 272.2327, Y 58.9340, Z -2.1667, A 0.000, B 0.000, C 0.000 }
gfCNCPoint1[29548] = {X 272.2327, Y 58.0000, Z -2.1667, A 0.000, B 0.000, C 0.000 }
gfCNCPoint1[29549] = {X 272.3330, Y 57.1099, Z -2.1667, A 0.000, B 0.000, C 0.000 }
gfCNCPoint1[29550] = {X 272.6288, Y 56.2645, Z -2.1667, A 0.000, B 0.000, C 0.000 }
gfCNCPoint1[29551] = {X 273.1054, Y 55.5060, Z -2.1667, A 0.000, B 0.000, C 0.000 }
gfCNCPoint1[29552] = {X 273.7387, Y 54.8727, Z -2.1667, A 0.000, B 0.000, C 0.000 }
gfCNCPoint1[29553] = {X 274.4972, Y 54.3961, Z -2.1667, A 0.000, B 0.000, C 0.000 }
gfCNCPoint1[29554] = {X 275.3426, Y 54.1003, Z -2.1667, A 0.000, B 0.000, C 0.000 }
gfCNCPoint1[29555] = {X 276.2327, Y 54.0000, Z -2.1667, A 0.000, B 0.000, C 0.000 }
gfCNCPoint1[29556] = {X 292.7731, Y 54.0000, Z -2.1667, A 0.000, B 0.000, C 0.000 }
gfCNCPoint1[29557] = {X 293.6632, Y 54.1003, Z -2.1667, A 0.000, B 0.000, C 0.000 }
gfCNCPoint1[29558] = {X 294.5086, Y 54.3961, Z -2.1667, A 0.000, B 0.000, C 0.000 }
gfCNCPoint1[29559] = {X 295.2670, Y 54.8727, Z -2.1667, A 0.000, B 0.000, C 0.000 }
gfCNCPoint1[29560] = {X 295.9004, Y 55.5060, Z -2.1667, A 0.000, B 0.000, C 0.000 }
gfCNCPoint1[29561] = {X 296.3770, Y 56.2645, Z -2.1667, A 0.000, B 0.000, C 0.000 }
gfCNCPoint1[29562] = {X 296.6728, Y 57.1099, Z -2.1667, A 0.000, B 0.000, C 0.000 }
gfCNCPoint1[29563] = {X 296.7731, Y 58.0000, Z -2.1667, A 0.000, B 0.000, C 0.000 }
gfCNCPoint1[29564] = {X 296.7731, Y 58.9341, Z -2.1667, A 0.000, B 0.000, C 0.000 }
gfCNCPoint1[29565] = {X 296.6596, Y 59.8685, Z -2.1667, A 0.000, B 0.000, C 0.000 }
gfCNCPoint1[29566] = {X 296.3317, Y 60.7508, Z -2.1667, A 0.000, B 0.000, C 0.000 }
gfCNCPoint1[29567] = {X 295.8075, Y 61.5326, Z -2.1667, A 0.000, B 0.000, C 0.000 }
gfCNCPoint1[29568] = {X 295.1158, Y 62.1710, Z -2.1667, A 0.000, B 0.000, C 0.000 }
gfCNCPoint1[29569] = {X 294.2945, Y 62.6309, Z -2.1667, A 0.000, B 0.000, C 0.000 }
gfCNCPoint1[29570] = {X 293.3888, Y 62.8870, Z -2.1667, A 0.000, B 0.000, C 0.000 }
gfCNCPoint1[29571] = {X 293.2323, Y 62.9088, Z -2.1667, A 0.000, B 0.000, C 0.000 }
gfCNCPoint1[29572] = {X 293.0752, Y 62.9244, Z -2.1667, A 0.000, B 0.000, C 0.000 }
gfCNCPoint1[29573] = {X 293.0518, Y 63.1540, Z -2.1667, A 0.000, B 0.000, C 0.000 }
gfCNCPoint1[29574] = {X 293.0518, Y 92.9237, Z -2.1667, A 0.000, B 0.000, C 0.000 }
gfCNCPoint1[29575] = {X 293.0752, Y 93.0681, Z -2.1667, A 0.000, B 0.000, C 0.000 }
gfCNCPoint1[29576] = {X 293.2317, Y 93.0843, Z -2.1667, A 0.000, B 0.000, C 0.000 }
gfCNCPoint1[29577] = {X 293.3876, Y 93.1065, Z -2.1667, A 0.000, B 0.000, C 0.000 }
gfCNCPoint1[29578] = {X 294.2931, Y 93.3652, Z -2.1667, A 0.000, B 0.000, C 0.000 }
gfCNCPoint1[29579] = {X 295.1140, Y 93.8269, Z -2.1667, A 0.000, B 0.000, C 0.000 }
gfCNCPoint1[29580] = {X 295.8054, Y 94.4663, Z -2.1667, A 0.000, B 0.000, C 0.000 }
gfCNCPoint1[29581] = {X 296.3297, Y 95.2487, Z -2.1667, A 0.000, B 0.000, C 0.000 }
gfCNCPoint1[29582] = {X 296.6582, Y 96.1313, Z -2.1667, A 0.000, B 0.000, C 0.000 }
gfCNCPoint1[29583] = {X 296.7731, Y 97.0661, Z -2.1667, A 0.000, B 0.000, C 0.000 }
gfCNCPoint1[29584] = {X 296.7731, Y 98.0000, Z -2.1667, A 0.000, B 0.000, C 0.000 }
gfCNCPoint1[29585] = {X 296.6728, Y 98.8901, Z -2.1667, A 0.000, B 0.000, C 0.000 }
gfCNCPoint1[29586] = {X 296.3770, Y 99.7355, Z -2.1667, A 0.000, B 0.000, C 0.000 }
gfCNCPoint1[29587] = {X 295.9004, Y 100.4940, Z -2.1667, A 0.000, B 0.000, C 0.000 }
gfCNCPoint1[29588] = {X 295.2670, Y 101.1273, Z -2.1667, A 0.000, B 0.000, C 0.000 }
gfCNCPoint1[29589] = {X 294.5086, Y 101.6039, Z -2.1667, A 0.000, B 0.000, C 0.000 }
gfCNCPoint1[29590] = {X 293.6632, Y 101.8997, Z -2.1667, A 0.000, B 0.000, C 0.000 }
gfCNCPoint1[29591] = {X 292.7731, Y 102.0000, Z -2.1667, A 0.000, B 0.000, C 0.000 }
gfCNCPoint1[29592] = {X 276.2327, Y 102.0000, Z -2.1667, A 0.000, B 0.000, C 0.000 }
gfCNCPoint1[29593] = {X 275.3426, Y 101.8997, Z -2.1667, A 0.000, B 0.000, C 0.000 }
gfCNCPoint1[29594] = {X 274.4972, Y 101.6039, Z -2.1667, A 0.000, B 0.000, C 0.000 }
gfCNCPoint1[29595] = {X 273.7387, Y 101.1273, Z -2.1667, A 0.000, B 0.000, C 0.000 }
gfCNCPoint1[29596] = {X 273.1054, Y 100.4940, Z -2.1667, A 0.000, B 0.000, C 0.000 }
gfCNCPoint1[29597] = {X 272.6288, Y 99.7355, Z -2.1667, A 0.000, B 0.000, C 0.000 }
gfCNCPoint1[29598] = {X 272.3330, Y 98.8901, Z -2.1667, A 0.000, B 0.000, C 0.000 }
gfCNCPoint1[29599] = {X 272.2327, Y 98.0000, Z -2.1667, A 0.000, B 0.000, C 0.000 }
gfCNCPoint1[29600] = {X 272.2329, Y 97.0232, Z -2.1667, A 0.000, B 0.000, C 0.000 }
gfCNCPoint1[29601] = {X 272.3321, Y 96.1797, Z -2.1667, A 0.000, B 0.000, C 0.000 }
gfCNCPoint1[29602] = {X 272.6072, Y 95.3761, Z -2.1667, A 0.000, B 0.000, C 0.000 }
gfCNCPoint1[29603] = {X 273.0457, Y 94.6486, Z -2.1667, A 0.000, B 0.000, C 0.000 }
gfCNCPoint1[29604] = {X 273.6280, Y 94.0302, Z -2.1667, A 0.000, B 0.000, C 0.000 }
gfCNCPoint1[29605] = {X 274.3277, Y 93.5487, Z -2.1667, A 0.000, B 0.000, C 0.000 }
gfCNCPoint1[29606] = {X 275.1133, Y 93.2258, Z -2.1667, A 0.000, B 0.000, C 0.000 }
gfCNCPoint1[29607] = {X 275.9494, Y 93.0760, Z -2.1667, A 0.000, B 0.000, C 0.000 }
gfCNCPoint1[29608] = {X 275.9494, Y 85.3767, Z -2.1667, A 0.000, B 0.000, C 0.000 }
gfCNCPoint1[29609] = {X 262.6059, Y 80.1460, Z -2.1667, A 0.000, B 0.000, C 0.000 }
gfCNCPoint1[29610] = {X 262.1037, Y 80.4620, Z -2.1667, A 0.000, B 0.000, C 0.000 }
gfCNCPoint1[29611] = {X 237.4745, Y 96.4149, Z -2.1667, A 0.000, B 0.000, C 0.000 }
gfCNCPoint1[29612] = {X 237.4798, Y 97.0659, Z -2.1667, A 0.000, B 0.000, C 0.000 }
gfCNCPoint1[29613] = {X 237.4798, Y 98.0000, Z -2.1667, A 0.000, B 0.000, C 0.000 }
gfCNCPoint1[29614] = {X 237.3795, Y 98.8901, Z -2.1667, A 0.000, B 0.000, C 0.000 }
gfCNCPoint1[29615] = {X 237.0837, Y 99.7355, Z -2.1667, A 0.000, B 0.000, C 0.000 }
gfCNCPoint1[29616] = {X 236.6071, Y 100.4940, Z -2.1667, A 0.000, B 0.000, C 0.000 }
gfCNCPoint1[29617] = {X 235.9737, Y 101.1273, Z -2.1667, A 0.000, B 0.000, C 0.000 }
gfCNCPoint1[29618] = {X 235.2153, Y 101.6039, Z -2.1667, A 0.000, B 0.000, C 0.000 }
gfCNCPoint1[29619] = {X 234.3699, Y 101.8997, Z -2.1667, A 0.000, B 0.000, C 0.000 }
gfCNCPoint1[29620] = {X 233.4798, Y 102.0000, Z -2.1667, A 0.000, B 0.000, C 0.000 }
gfCNCPoint1[29621] = {X 214.1790, Y 102.0000, Z -2.1667, A 0.000, B 0.000, C 0.000 }
gfCNCPoint1[29622] = {X 213.7859, Y 101.9806, Z -2.1667, A 0.000, B 0.000, C 0.000 }
gfCNCPoint1[29623] = {X 213.3966, Y 101.9227, Z -2.1667, A 0.000, B 0.000, C 0.000 }
gfCNCPoint1[29624] = {X 213.0072, Y 101.9806, Z -2.1667, A 0.000, B 0.000, C 0.000 }
gfCNCPoint1[29625] = {X 212.6141, Y 102.0000, Z -2.1667, A 0.000, B 0.000, C 0.000 }
gfCNCPoint1[29626] = {X 194.9870, Y 102.0000, Z -2.1667, A 0.000, B 0.000, C 0.000 }
gfCNCPoint1[29627] = {X 194.0969, Y 101.8997, Z -2.1667, A 0.000, B 0.000, C 0.000 }
gfCNCPoint1[29628] = {X 193.2514, Y 101.6039, Z -2.1667, A 0.000, B 0.000, C 0.000 }
gfCNCPoint1[29629] = {X 192.4930, Y 101.1273, Z -2.1667, A 0.000, B 0.000, C 0.000 }
gfCNCPoint1[29630] = {X 191.8596, Y 100.4940, Z -2.1667, A 0.000, B 0.000, C 0.000 }
gfCNCPoint1[29631] = {X 191.3831, Y 99.7355, Z -2.1667, A 0.000, B 0.000, C 0.000 }
gfCNCPoint1[29632] = {X 191.0872, Y 98.8901, Z -2.1667, A 0.000, B 0.000, C 0.000 }
gfCNCPoint1[29633] = {X 190.9870, Y 98.0000, Z -2.1667, A 0.000, B 0.000, C 0.000 }
gfCNCPoint1[29634] = {X 190.9870, Y 97.0659, Z -2.1667, A 0.000, B 0.000, C 0.000 }
gfCNCPoint1[29635] = {X 191.0804, Y 96.2066, Z -2.1667, A 0.000, B 0.000, C 0.000 }
gfCNCPoint1[29636] = {X 191.3562, Y 95.3874, Z -2.1667, A 0.000, B 0.000, C 0.000 }
gfCNCPoint1[29637] = {X 191.8015, Y 94.6466, Z -2.1667, A 0.000, B 0.000, C 0.000 }
gfCNCPoint1[29638] = {X 191.8852, Y 94.5402, Z -2.1667, A 0.000, B 0.000, C 0.000 }
gfCNCPoint1[29639] = {X 191.9725, Y 94.4367, Z -2.1667, A 0.000, B 0.000, C 0.000 }
gfCNCPoint1[29640] = {X 192.0152, Y 94.3936, Z -2.1667, A 0.000, B 0.000, C 0.000 }
gfCNCPoint1[29641] = {X 188.7055, Y 90.7802, Z -2.1667, A 0.000, B 0.000, C 0.000 }
gfCNCPoint1[29642] = {X 149.9476, Y 90.7802, Z -2.1667, A 0.000, B 0.000, C 0.000 }
gfCNCPoint1[29643] = {X 146.7184, Y 94.3578, Z -2.1667, A 0.000, B 0.000, C 0.000 }
gfCNCPoint1[29644] = {X 147.1681, Y 94.9491, Z -2.1667, A 0.000, B 0.000, C 0.000 }
gfCNCPoint1[29645] = {X 147.5016, Y 95.6129, Z -2.1667, A 0.000, B 0.000, C 0.000 }
gfCNCPoint1[29646] = {X 147.7076, Y 96.3267, Z -2.1667, A 0.000, B 0.000, C 0.000 }
gfCNCPoint1[29647] = {X 147.7791, Y 97.0661, Z -2.1667, A 0.000, B 0.000, C 0.000 }
gfCNCPoint1[29648] = {X 147.7791, Y 98.0000, Z -2.1667, A 0.000, B 0.000, C 0.000 }
gfCNCPoint1[29649] = {X 147.6788, Y 98.8901, Z -2.1667, A 0.000, B 0.000, C 0.000 }
gfCNCPoint1[29650] = {X 147.3830, Y 99.7355, Z -2.1667, A 0.000, B 0.000, C 0.000 }
gfCNCPoint1[29651] = {X 146.9064, Y 100.4940, Z -2.1667, A 0.000, B 0.000, C 0.000 }
gfCNCPoint1[29652] = {X 146.2731, Y 101.1273, Z -2.1667, A 0.000, B 0.000, C 0.000 }
gfCNCPoint1[29653] = {X 145.5146, Y 101.6039, Z -2.1667, A 0.000, B 0.000, C 0.000 }
gfCNCPoint1[29654] = {X 144.6692, Y 101.8997, Z -2.1667, A 0.000, B 0.000, C 0.000 }
gfCNCPoint1[29655] = {X 143.7791, Y 102.0000, Z -2.1667, A 0.000, B 0.000, C 0.000 }
gfCNCPoint1[29656] = {X 125.0000, Y 102.0000, Z -2.1667, A 0.000, B 0.000, C 0.000 }
gfCNCPoint1[29657] = {X 124.1099, Y 101.8997, Z -2.1667, A 0.000, B 0.000, C 0.000 }
gfCNCPoint1[29658] = {X 123.2645, Y 101.6039, Z -2.1667, A 0.000, B 0.000, C 0.000 }
gfCNCPoint1[29659] = {X 122.5060, Y 101.1273, Z -2.1667, A 0.000, B 0.000, C 0.000 }
gfCNCPoint1[29660] = {X 121.8727, Y 100.4940, Z -2.1667, A 0.000, B 0.000, C 0.000 }
gfCNCPoint1[29661] = {X 121.3961, Y 99.7355, Z -2.1667, A 0.000, B 0.000, C 0.000 }
gfCNCPoint1[29662] = {X 121.1003, Y 98.8901, Z -2.1667, A 0.000, B 0.000, C 0.000 }
gfCNCPoint1[29663] = {X 121.0000, Y 98.0000, Z -2.1667, A 0.000, B 0.000, C 0.000 }
gfCNCPoint1[29664] = {X 121.0000, Y 97.0659, Z -2.1667, A 0.000, B 0.000, C 0.000 }
gfCNCPoint1[29665] = {X 121.0981, Y 96.1853, Z -2.1667, A 0.000, B 0.000, C 0.000 }
gfCNCPoint1[29666] = {X 121.3877, Y 95.3479, Z -2.1667, A 0.000, B 0.000, C 0.000 }
gfCNCPoint1[29667] = {X 121.8546, Y 94.5948, Z -2.1667, A 0.000, B 0.000, C 0.000 }
gfCNCPoint1[29668] = {X 122.4758, Y 93.9629, Z -2.1667, A 0.000, B 0.000, C 0.000 }
gfCNCPoint1[29669] = {X 123.2209, Y 93.4834, Z -2.1667, A 0.000, B 0.000, C 0.000 }
gfCNCPoint1[29670] = {X 124.0533, Y 93.1796, Z -2.1667, A 0.000, B 0.000, C 0.000 }
gfCNCPoint1[29671] = {X 124.9321, Y 93.0665, Z -2.1667, A 0.000, B 0.000, C 0.000 }
gfCNCPoint1[29672] = {X 124.9750, Y 93.0390, Z -2.1667, A 0.000, B 0.000, C 0.000 }
gfCNCPoint1[29673] = {X 125.4940, Y 92.9620, Z -2.1667, A 0.000, B 0.000, C 0.000 }
gfCNCPoint1[29674] = {X 126.3824, Y 92.8101, Z -2.1667, A 0.000, B 0.000, C 0.000 }
gfCNCPoint1[29675] = {X 127.2581, Y 92.5970, Z -2.1667, A 0.000, B 0.000, C 0.000 }
gfCNCPoint1[29676] = {X 128.5217, Y 91.4098, Z -2.1667, A 0.000, B 0.000, C 0.000 }
gfCNCPoint1[29677] = {X 129.7176, Y 90.1544, Z -2.1667, A 0.000, B 0.000, C 0.000 }
gfCNCPoint1[29678] = {X 133.8038, Y 85.6595, Z -2.1667, A 0.000, B 0.000, C 0.000 }
gfCNCPoint1[29679] = {X 140.9144, Y 77.8536, Z -2.1667, A 0.000, B 0.000, C 0.000 }
gfCNCPoint1[29680] = {X 137.8982, Y 75.1061, Z -2.1667, A 0.000, B 0.000, C 0.000 }
gfCNCPoint1[29681] = {X 137.8982, Y 75.1061, Z 0.8333, A 0.000, B 0.000, C 0.000 }
gfCNCPoint1[29682] = {X 137.8982, Y 75.1061, Z 11.0000, A 0.000, B 0.000, C 0.000 }
gfCNCPoint1[29683] = {X 167.3809, Y 20.2812, Z 11.0000, A 0.000, B 0.000, C 0.000 }
gfCNCPoint1[29684] = {X 167.3809, Y 20.2812, Z 0.8333, A 0.000, B 0.000, C 0.000 }
gfCNCPoint1[29685] = {X 167.3809, Y 20.2812, Z -2.1667, A 0.000, B 0.000, C 0.000 }
gfCNCPoint1[29686] = {X 171.1581, Y 18.7388, Z -2.1667, A 0.000, B 0.000, C 0.000 }
gfCNCPoint1[29687] = {X 169.8405, Y 15.5121, Z -2.1667, A 0.000, B 0.000, C 0.000 }
gfCNCPoint1[29688] = {X 169.5912, Y 14.6607, Z -2.1667, A 0.000, B 0.000, C 0.000 }
gfCNCPoint1[29689] = {X 169.5212, Y 13.7764, Z -2.1667, A 0.000, B 0.000, C 0.000 }
gfCNCPoint1[29690] = {X 169.6332, Y 12.8964, Z -2.1667, A 0.000, B 0.000, C 0.000 }
gfCNCPoint1[29691] = {X 169.9226, Y 12.0578, Z -2.1667, A 0.000, B 0.000, C 0.000 }
gfCNCPoint1[29692] = {X 170.3773, Y 11.2960, Z -2.1667, A 0.000, B 0.000, C 0.000 }
gfCNCPoint1[29693] = {X 170.9779, Y 10.6432, Z -2.1667, A 0.000, B 0.000, C 0.000 }
gfCNCPoint1[29694] = {X 171.6992, Y 10.1268, Z -2.1667, A 0.000, B 0.000, C 0.000 }
gfCNCPoint1[29695] = {X 172.3295, Y 9.7674, Z -2.1667, A 0.000, B 0.000, C 0.000 }
gfCNCPoint1[29696] = {X 173.2114, Y 9.3960, Z -2.1667, A 0.000, B 0.000, C 0.000 }
gfCNCPoint1[29697] = {X 174.1534, Y 9.2278, Z -2.1667, A 0.000, B 0.000, C 0.000 }
gfCNCPoint1[29698] = {X 175.1093, Y 9.2711, Z -2.1667, A 0.000, B 0.000, C 0.000 }
gfCNCPoint1[29699] = {X 176.0323, Y 9.5238, Z -2.1667, A 0.000, B 0.000, C 0.000 }
gfCNCPoint1[29700] = {X 178.2250, Y 8.6013, Z -2.1667, A 0.000, B 0.000, C 0.000 }
gfCNCPoint1[29701] = {X 180.4990, Y 7.9027, Z -2.1667, A 0.000, B 0.000, C 0.000 }
gfCNCPoint1[29702] = {X 182.8314, Y 7.4350, Z -2.1667, A 0.000, B 0.000, C 0.000 }
gfCNCPoint1[29703] = {X 185.1989, Y 7.2029, Z -2.1667, A 0.000, B 0.000, C 0.000 }
gfCNCPoint1[29704] = {X 187.5778, Y 7.2087, Z -2.1667, A 0.000, B 0.000, C 0.000 }
gfCNCPoint1[29705] = {X 189.9442, Y 7.4523, Z -2.1667, A 0.000, B 0.000, C 0.000 }
gfCNCPoint1[29706] = {X 191.7013, Y 7.8139, Z -2.1667, A 0.000, B 0.000, C 0.000 }
gfCNCPoint1[29707] = {X 193.4121, Y 8.3540, Z -2.1667, A 0.000, B 0.000, C 0.000 }
gfCNCPoint1[29708] = {X 195.0584, Y 9.0667, Z -2.1667, A 0.000, B 0.000, C 0.000 }
gfCNCPoint1[29709] = {X 196.6228, Y 9.9447, Z -2.1667, A 0.000, B 0.000, C 0.000 }
gfCNCPoint1[29710] = {X 198.0890, Y 10.9785, Z -2.1667, A 0.000, B 0.000, C 0.000 }
gfCNCPoint1[29711] = {X 199.1485, Y 11.9219, Z -2.1667, A 0.000, B 0.000, C 0.000 }
gfCNCPoint1[29712] = {X 200.0994, Y 12.9747, Z -2.1667, A 0.000, B 0.000, C 0.000 }
gfCNCPoint1[29713] = {X 200.9304, Y 14.1245, Z -2.1667, A 0.000, B 0.000, C 0.000 }
gfCNCPoint1[29714] = {X 201.6317, Y 15.3578, Z -2.1667, A 0.000, B 0.000, C 0.000 }
gfCNCPoint1[29715] = {X 202.1950, Y 16.6598, Z -2.1667, A 0.000, B 0.000, C 0.000 }
gfCNCPoint1[29716] = {X 202.6692, Y 18.3162, Z -2.1667, A 0.000, B 0.000, C 0.000 }
gfCNCPoint1[29717] = {X 202.9507, Y 20.0159, Z -2.1667, A 0.000, B 0.000, C 0.000 }
gfCNCPoint1[29718] = {X 203.0357, Y 21.7367, Z -2.1667, A 0.000, B 0.000, C 0.000 }
gfCNCPoint1[29719] = {X 202.9231, Y 23.4559, Z -2.1667, A 0.000, B 0.000, C 0.000 }
gfCNCPoint1[29720] = {X 202.6145, Y 25.1510, Z -2.1667, A 0.000, B 0.000, C 0.000 }
gfCNCPoint1[29721] = {X 202.1727, Y 26.5971, Z -2.1667, A 0.000, B 0.000, C 0.000 }
gfCNCPoint1[29722] = {X 201.5480, Y 27.9741, Z -2.1667, A 0.000, B 0.000, C 0.000 }
gfCNCPoint1[29723] = {X 200.7508, Y 29.2589, Z -2.1667, A 0.000, B 0.000, C 0.000 }
gfCNCPoint1[29724] = {X 199.7944, Y 30.4302, Z -2.1667, A 0.000, B 0.000, C 0.000 }
gfCNCPoint1[29725] = {X 198.6949, Y 31.4681, Z -2.1667, A 0.000, B 0.000, C 0.000 }
gfCNCPoint1[29726] = {X 199.4965, Y 31.8093, Z -2.1667, A 0.000, B 0.000, C 0.000 }
gfCNCPoint1[29727] = {X 200.2133, Y 32.3044, Z -2.1667, A 0.000, B 0.000, C 0.000 }
gfCNCPoint1[29728] = {X 200.8163, Y 32.9332, Z -2.1667, A 0.000, B 0.000, C 0.000 }
gfCNCPoint1[29729] = {X 201.2808, Y 33.6702, Z -2.1667, A 0.000, B 0.000, C 0.000 }
gfCNCPoint1[29730] = {X 204.3222, Y 39.9530, Z -2.1667, A 0.000, B 0.000, C 0.000 }
gfCNCPoint1[29731] = {X 204.6427, Y 40.8622, Z -2.1667, A 0.000, B 0.000, C 0.000 }
gfCNCPoint1[29732] = {X 204.7537, Y 41.8197, Z -2.1667, A 0.000, B 0.000, C 0.000 }
gfCNCPoint1[29733] = {X 204.6496, Y 42.7781, Z -2.1667, A 0.000, B 0.000, C 0.000 }
gfCNCPoint1[29734] = {X 204.3355, Y 43.6895, Z -2.1667, A 0.000, B 0.000, C 0.000 }
gfCNCPoint1[29735] = {X 203.8272, Y 44.5085, Z -2.1667, A 0.000, B 0.000, C 0.000 }
gfCNCPoint1[29736] = {X 203.1499, Y 45.1945, Z -2.1667, A 0.000, B 0.000, C 0.000 }
gfCNCPoint1[29737] = {X 202.6135, Y 45.6282, Z -2.1667, A 0.000, B 0.000, C 0.000 }
gfCNCPoint1[29738] = {X 201.9087, Y 46.0914, Z -2.1667, A 0.000, B 0.000, C 0.000 }
gfCNCPoint1[29739] = {X 201.1276, Y 46.4095, Z -2.1667, A 0.000, B 0.000, C 0.000 }
gfCNCPoint1[29740] = {X 200.2997, Y 46.5703, Z -2.1667, A 0.000, B 0.000, C 0.000 }
gfCNCPoint1[29741] = {X 199.4564, Y 46.5678, Z -2.1667, A 0.000, B 0.000, C 0.000 }
gfCNCPoint1[29742] = {X 198.6294, Y 46.4021, Z -2.1667, A 0.000, B 0.000, C 0.000 }
gfCNCPoint1[29743] = {X 196.8919, Y 47.3243, Z -2.1667, A 0.000, B 0.000, C 0.000 }
gfCNCPoint1[29744] = {X 195.0953, Y 48.1251, Z -2.1667, A 0.000, B 0.000, C 0.000 }
gfCNCPoint1[29745] = {X 193.2478, Y 48.8006, Z -2.1667, A 0.000, B 0.000, C 0.000 }
gfCNCPoint1[29746] = {X 191.3584, Y 49.3478, Z -2.1667, A 0.000, B 0.000, C 0.000 }
gfCNCPoint1[29747] = {X 189.4153, Y 49.7415, Z -2.1667, A 0.000, B 0.000, C 0.000 }
gfCNCPoint1[29748] = {X 187.4452, Y 49.9638, Z -2.1667, A 0.000, B 0.000, C 0.000 }
gfCNCPoint1[29749] = {X 185.4633, Y 50.0129, Z -2.1667, A 0.000, B 0.000, C 0.000 }
gfCNCPoint1[29750] = {X 183.4846, Y 49.8886, Z -2.1667, A 0.000, B 0.000, C 0.000 }
gfCNCPoint1[29751] = {X 181.5244, Y 49.5917, Z -2.1667, A 0.000, B 0.000, C 0.000 }
gfCNCPoint1[29752] = {X 179.6379, Y 49.1201, Z -2.1667, A 0.000, B 0.000, C 0.000 }
gfCNCPoint1[29753] = {X 177.8176, Y 48.4367, Z -2.1667, A 0.000, B 0.000, C 0.000 }
gfCNCPoint1[29754] = {X 176.0869, Y 47.5502, Z -2.1667, A 0.000, B 0.000, C 0.000 }
gfCNCPoint1[29755] = {X 174.4685, Y 46.4723, Z -2.1667, A 0.000, B 0.000, C 0.000 }
gfCNCPoint1[29756] = {X 173.2359, Y 45.4318, Z -2.1667, A 0.000, B 0.000, C 0.000 }
gfCNCPoint1[29757] = {X 172.1389, Y 44.2492, Z -2.1667, A 0.000, B 0.000, C 0.000 }
gfCNCPoint1[29758] = {X 171.1940, Y 42.9418, Z -2.1667, A 0.000, B 0.000, C 0.000 }
gfCNCPoint1[29759] = {X 170.4152, Y 41.5292, Z -2.1667, A 0.000, B 0.000, C 0.000 }
gfCNCPoint1[29760] = {X 169.8141, Y 40.0323, Z -2.1667, A 0.000, B 0.000, C 0.000 }
gfCNCPoint1[29761] = {X 169.3995, Y 38.4734, Z -2.1667, A 0.000, B 0.000, C 0.000 }
gfCNCPoint1[29762] = {X 169.1776, Y 36.8757, Z -2.1667, A 0.000, B 0.000, C 0.000 }
gfCNCPoint1[29763] = {X 169.0934, Y 35.0418, Z -2.1667, A 0.000, B 0.000, C 0.000 }
gfCNCPoint1[29764] = {X 169.2394, Y 33.2119, Z -2.1667, A 0.000, B 0.000, C 0.000 }
gfCNCPoint1[29765] = {X 169.6134, Y 31.4146, Z -2.1667, A 0.000, B 0.000, C 0.000 }
gfCNCPoint1[29766] = {X 170.2096, Y 29.6784, Z -2.1667, A 0.000, B 0.000, C 0.000 }
gfCNCPoint1[29767] = {X 170.8486, Y 28.3713, Z -2.1667, A 0.000, B 0.000, C 0.000 }
gfCNCPoint1[29768] = {X 171.6566, Y 27.1613, Z -2.1667, A 0.000, B 0.000, C 0.000 }
gfCNCPoint1[29769] = {X 172.6190, Y 26.0702, Z -2.1667, A 0.000, B 0.000, C 0.000 }
gfCNCPoint1[29770] = {X 173.7186, Y 25.1174, Z -2.1667, A 0.000, B 0.000, C 0.000 }
gfCNCPoint1[29771] = {X 174.9357, Y 24.3202, Z -2.1667, A 0.000, B 0.000, C 0.000 }
gfCNCPoint1[29772] = {X 174.1528, Y 23.9326, Z -2.1667, A 0.000, B 0.000, C 0.000 }
gfCNCPoint1[29773] = {X 173.4639, Y 23.3954, Z -2.1667, A 0.000, B 0.000, C 0.000 }
gfCNCPoint1[29774] = {X 172.8972, Y 22.7306, Z -2.1667, A 0.000, B 0.000, C 0.000 }
gfCNCPoint1[29775] = {X 172.4758, Y 21.9655, Z -2.1667, A 0.000, B 0.000, C 0.000 }
gfCNCPoint1[29776] = {X 171.1581, Y 18.7388, Z -2.1667, A 0.000, B 0.000, C 0.000 }
gfCNCPoint1[29777] = {X 167.4550, Y 20.2510, Z -2.1667, A 0.000, B 0.000, C 0.000 }
gfCNCPoint1[29778] = {X 171.2322, Y 18.7085, Z -2.1667, A 0.000, B 0.000, C 0.000 }
gfCNCPoint1[29779] = {X 169.9145, Y 15.4818, Z -2.1667, A 0.000, B 0.000, C 0.000 }
gfCNCPoint1[29780] = {X 169.6699, Y 14.6462, Z -2.1667, A 0.000, B 0.000, C 0.000 }
gfCNCPoint1[29781] = {X 169.6011, Y 13.7783, Z -2.1667, A 0.000, B 0.000, C 0.000 }
gfCNCPoint1[29782] = {X 169.7111, Y 12.9146, Z -2.1667, A 0.000, B 0.000, C 0.000 }
gfCNCPoint1[29783] = {X 169.9952, Y 12.0915, Z -2.1667, A 0.000, B 0.000, C 0.000 }
gfCNCPoint1[29784] = {X 170.4414, Y 11.3439, Z -2.1667, A 0.000, B 0.000, C 0.000 }
gfCNCPoint1[29785] = {X 171.0309, Y 10.7031, Z -2.1667, A 0.000, B 0.000, C 0.000 }
gfCNCPoint1[29786] = {X 171.7389, Y 10.1963, Z -2.1667, A 0.000, B 0.000, C 0.000 }
gfCNCPoint1[29787] = {X 172.3689, Y 9.8371, Z -2.1667, A 0.000, B 0.000, C 0.000 }
gfCNCPoint1[29788] = {X 173.2427, Y 9.4701, Z -2.1667, A 0.000, B 0.000, C 0.000 }
gfCNCPoint1[29789] = {X 174.1763, Y 9.3065, Z -2.1667, A 0.000, B 0.000, C 0.000 }
gfCNCPoint1[29790] = {X 175.1229, Y 9.3543, Z -2.1667, A 0.000, B 0.000, C 0.000 }
gfCNCPoint1[29791] = {X 176.0352, Y 9.6112, Z -2.1667, A 0.000, B 0.000, C 0.000 }
gfCNCPoint1[29792] = {X 178.2247, Y 8.6865, Z -2.1667, A 0.000, B 0.000, C 0.000 }
gfCNCPoint1[29793] = {X 180.4958, Y 7.9860, Z -2.1667, A 0.000, B 0.000, C 0.000 }
gfCNCPoint1[29794] = {X 182.8258, Y 7.5168, Z -2.1667, A 0.000, B 0.000, C 0.000 }
gfCNCPoint1[29795] = {X 185.1910, Y 7.2834, Z -2.1667, A 0.000, B 0.000, C 0.000 }
gfCNCPoint1[29796] = {X 187.5678, Y 7.2883, Z -2.1667, A 0.000, B 0.000, C 0.000 }
gfCNCPoint1[29797] = {X 189.9320, Y 7.5314, Z -2.1667, A 0.000, B 0.000, C 0.000 }
gfCNCPoint1[29798] = {X 191.6811, Y 7.8914, Z -2.1667, A 0.000, B 0.000, C 0.000 }
gfCNCPoint1[29799] = {X 193.3841, Y 8.4289, Z -2.1667, A 0.000, B 0.000, C 0.000 }
gfCNCPoint1[29800] = {X 195.0228, Y 9.1384, Z -2.1667, A 0.000, B 0.000, C 0.000 }
gfCNCPoint1[29801] = {X 196.5802, Y 10.0123, Z -2.1667, A 0.000, B 0.000, C 0.000 }
gfCNCPoint1[29802] = {X 198.0396, Y 11.0414, Z -2.1667, A 0.000, B 0.000, C 0.000 }
gfCNCPoint1[29803] = {X 199.3393, Y 12.2308, Z -2.1667, A 0.000, B 0.000, C 0.000 }
gfCNCPoint1[29804] = {X 200.4659, Y 13.5854, Z -2.1667, A 0.000, B 0.000, C 0.000 }
gfCNCPoint1[29805] = {X 201.3985, Y 15.0802, Z -2.1667, A 0.000, B 0.000, C 0.000 }
gfCNCPoint1[29806] = {X 202.1200, Y 16.6876, Z -2.1667, A 0.000, B 0.000, C 0.000 }
gfCNCPoint1[29807] = {X 202.5914, Y 18.3349, Z -2.1667, A 0.000, B 0.000, C 0.000 }
gfCNCPoint1[29808] = {X 202.8712, Y 20.0254, Z -2.1667, A 0.000, B 0.000, C 0.000 }
gfCNCPoint1[29809] = {X 202.9557, Y 21.7368, Z -2.1667, A 0.000, B 0.000, C 0.000 }
gfCNCPoint1[29810] = {X 202.8437, Y 23.4466, Z -2.1667, A 0.000, B 0.000, C 0.000 }
gfCNCPoint1[29811] = {X 202.5366, Y 25.1324, Z -2.1667, A 0.000, B 0.000, C 0.000 }
gfCNCPoint1[29812] = {X 202.0872, Y 26.5970, Z -2.1667, A 0.000, B 0.000, C 0.000 }
gfCNCPoint1[29813] = {X 201.4488, Y 27.9896, Z -2.1667, A 0.000, B 0.000, C 0.000 }
gfCNCPoint1[29814] = {X 200.6327, Y 29.2861, Z -2.1667, A 0.000, B 0.000, C 0.000 }
gfCNCPoint1[29815] = {X 199.6529, Y 30.4639, Z -2.1667, A 0.000, B 0.000, C 0.000 }
gfCNCPoint1[29816] = {X 198.5266, Y 31.5024, Z -2.1667, A 0.000, B 0.000, C 0.000 }
gfCNCPoint1[29817] = {X 199.3583, Y 31.8262, Z -2.1667, A 0.000, B 0.000, C 0.000 }
gfCNCPoint1[29818] = {X 200.1037, Y 32.3170, Z -2.1667, A 0.000, B 0.000, C 0.000 }
gfCNCPoint1[29819] = {X 200.7299, Y 32.9529, Z -2.1667, A 0.000, B 0.000, C 0.000 }
gfCNCPoint1[29820] = {X 201.2091, Y 33.7058, Z -2.1667, A 0.000, B 0.000, C 0.000 }
gfCNCPoint1[29821] = {X 204.2502, Y 39.9879, Z -2.1667, A 0.000, B 0.000, C 0.000 }
gfCNCPoint1[29822] = {X 204.5648, Y 40.8802, Z -2.1667, A 0.000, B 0.000, C 0.000 }
gfCNCPoint1[29823] = {X 204.6737, Y 41.8200, Z -2.1667, A 0.000, B 0.000, C 0.000 }
gfCNCPoint1[29824] = {X 204.5715, Y 42.7606, Z -2.1667, A 0.000, B 0.000, C 0.000 }
gfCNCPoint1[29825] = {X 204.2633, Y 43.6551, Z -2.1667, A 0.000, B 0.000, C 0.000 }
gfCNCPoint1[29826] = {X 203.7643, Y 44.4590, Z -2.1667, A 0.000, B 0.000, C 0.000 }
gfCNCPoint1[29827] = {X 203.0996, Y 45.1323, Z -2.1667, A 0.000, B 0.000, C 0.000 }
gfCNCPoint1[29828] = {X 202.5632, Y 45.5659, Z -2.1667, A 0.000, B 0.000, C 0.000 }
gfCNCPoint1[29829] = {X 201.8654, Y 46.0238, Z -2.1667, A 0.000, B 0.000, C 0.000 }
gfCNCPoint1[29830] = {X 201.0916, Y 46.3367, Z -2.1667, A 0.000, B 0.000, C 0.000 }
gfCNCPoint1[29831] = {X 200.2715, Y 46.4926, Z -2.1667, A 0.000, B 0.000, C 0.000 }
gfCNCPoint1[29832] = {X 199.4369, Y 46.4854, Z -2.1667, A 0.000, B 0.000, C 0.000 }
gfCNCPoint1[29833] = {X 198.6197, Y 46.3154, Z -2.1667, A 0.000, B 0.000, C 0.000 }
gfCNCPoint1[29834] = {X 196.8804, Y 47.2410, Z -2.1667, A 0.000, B 0.000, C 0.000 }
gfCNCPoint1[29835] = {X 195.0814, Y 48.0444, Z -2.1667, A 0.000, B 0.000, C 0.000 }
gfCNCPoint1[29836] = {X 193.2312, Y 48.7219, Z -2.1667, A 0.000, B 0.000, C 0.000 }
gfCNCPoint1[29837] = {X 191.3388, Y 49.2702, Z -2.1667, A 0.000, B 0.000, C 0.000 }
gfCNCPoint1[29838] = {X 189.4026, Y 49.6625, Z -2.1667, A 0.000, B 0.000, C 0.000 }
gfCNCPoint1[29839] = {X 187.4395, Y 49.8840, Z -2.1667, A 0.000, B 0.000, C 0.000 }
gfCNCPoint1[29840] = {X 185.4645, Y 49.9329, Z -2.1667, A 0.000, B 0.000, C 0.000 }
gfCNCPoint1[29841] = {X 183.4929, Y 49.8090, Z -2.1667, A 0.000, B 0.000, C 0.000 }
gfCNCPoint1[29842] = {X 181.5396, Y 49.5131, Z -2.1667, A 0.000, B 0.000, C 0.000 }
gfCNCPoint1[29843] = {X 179.6619, Y 49.0438, Z -2.1667, A 0.000, B 0.000, C 0.000 }
gfCNCPoint1[29844] = {X 177.8500, Y 48.3635, Z -2.1667, A 0.000, B 0.000, C 0.000 }
gfCNCPoint1[29845] = {X 176.1273, Y 47.4812, Z -2.1667, A 0.000, B 0.000, C 0.000 }
gfCNCPoint1[29846] = {X 174.5165, Y 46.4083, Z -2.1667, A 0.000, B 0.000, C 0.000 }
gfCNCPoint1[29847] = {X 173.2911, Y 45.3740, Z -2.1667, A 0.000, B 0.000, C 0.000 }
gfCNCPoint1[29848] = {X 172.2007, Y 44.1983, Z -2.1667, A 0.000, B 0.000, C 0.000 }
gfCNCPoint1[29849] = {X 171.2614, Y 42.8986, Z -2.1667, A 0.000, B 0.000, C 0.000 }
gfCNCPoint1[29850] = {X 170.4872, Y 41.4943, Z -2.1667, A 0.000, B 0.000, C 0.000 }
gfCNCPoint1[29851] = {X 169.8897, Y 40.0063, Z -2.1667, A 0.000, B 0.000, C 0.000 }
gfCNCPoint1[29852] = {X 169.4777, Y 38.4566, Z -2.1667, A 0.000, B 0.000, C 0.000 }
gfCNCPoint1[29853] = {X 169.2573, Y 36.8682, Z -2.1667, A 0.000, B 0.000, C 0.000 }
gfCNCPoint1[29854] = {X 169.1733, Y 35.0441, Z -2.1667, A 0.000, B 0.000, C 0.000 }
gfCNCPoint1[29855] = {X 169.3185, Y 33.2237, Z -2.1667, A 0.000, B 0.000, C 0.000 }
gfCNCPoint1[29856] = {X 169.6905, Y 31.4359, Z -2.1667, A 0.000, B 0.000, C 0.000 }
gfCNCPoint1[29857] = {X 170.2836, Y 29.7088, Z -2.1667, A 0.000, B 0.000, C 0.000 }
gfCNCPoint1[29858] = {X 170.9357, Y 28.3805, Z -2.1667, A 0.000, B 0.000, C 0.000 }
gfCNCPoint1[29859] = {X 171.7635, Y 27.1540, Z -2.1667, A 0.000, B 0.000, C 0.000 }
gfCNCPoint1[29860] = {X 172.7515, Y 26.0523, Z -2.1667, A 0.000, B 0.000, C 0.000 }
gfCNCPoint1[29861] = {X 173.8809, Y 25.0963, Z -2.1667, A 0.000, B 0.000, C 0.000 }
gfCNCPoint1[29862] = {X 175.1306, Y 24.3038, Z -2.1667, A 0.000, B 0.000, C 0.000 }
gfCNCPoint1[29863] = {X 174.3089, Y 23.9337, Z -2.1667, A 0.000, B 0.000, C 0.000 }
gfCNCPoint1[29864] = {X 173.5840, Y 23.3983, Z -2.1667, A 0.000, B 0.000, C 0.000 }
gfCNCPoint1[29865] = {X 172.9886, Y 22.7218, Z -2.1667, A 0.000, B 0.000, C 0.000 }
gfCNCPoint1[29866] = {X 172.5496, Y 21.9347, Z -2.1667, A 0.000, B 0.000, C 0.000 }
gfCNCPoint1[29867] = {X 171.2322, Y 18.7085, Z -2.1667, A 0.000, B 0.000, C 0.000 }
gfCNCPoint1[29868] = {X 167.5291, Y 20.2207, Z -2.1667, A 0.000, B 0.000, C 0.000 }
gfCNCPoint1[29869] = {X 171.3062, Y 18.6783, Z -2.1667, A 0.000, B 0.000, C 0.000 }
gfCNCPoint1[29870] = {X 169.9886, Y 15.4516, Z -2.1667, A 0.000, B 0.000, C 0.000 }
gfCNCPoint1[29871] = {X 169.7252, Y 14.4911, Z -2.1667, A 0.000, B 0.000, C 0.000 }
gfCNCPoint1[29872] = {X 169.6977, Y 13.4955, Z -2.1667, A 0.000, B 0.000, C 0.000 }
gfCNCPoint1[29873] = {X 169.9076, Y 12.5218, Z -2.1667, A 0.000, B 0.000, C 0.000 }
gfCNCPoint1[29874] = {X 170.3429, Y 11.6260, Z -2.1667, A 0.000, B 0.000, C 0.000 }
gfCNCPoint1[29875] = {X 170.9787, Y 10.8594, Z -2.1667, A 0.000, B 0.000, C 0.000 }
gfCNCPoint1[29876] = {X 171.7785, Y 10.2658, Z -2.1667, A 0.000, B 0.000, C 0.000 }
gfCNCPoint1[29877] = {X 172.4082, Y 9.9068, Z -2.1667, A 0.000, B 0.000, C 0.000 }
gfCNCPoint1[29878] = {X 173.2740, Y 9.5443, Z -2.1667, A 0.000, B 0.000, C 0.000 }
gfCNCPoint1[29879] = {X 174.1991, Y 9.3853, Z -2.1667, A 0.000, B 0.000, C 0.000 }
gfCNCPoint1[29880] = {X 175.1362, Y 9.4376, Z -2.1667, A 0.000, B 0.000, C 0.000 }
gfCNCPoint1[29881] = {X 176.0378, Y 9.6988, Z -2.1667, A 0.000, B 0.000, C 0.000 }
gfCNCPoint1[29882] = {X 178.2241, Y 8.7719, Z -2.1667, A 0.000, B 0.000, C 0.000 }
gfCNCPoint1[29883] = {X 180.4925, Y 8.0695, Z -2.1667, A 0.000, B 0.000, C 0.000 }
gfCNCPoint1[29884] = {X 182.8200, Y 7.5985, Z -2.1667, A 0.000, B 0.000, C 0.000 }
gfCNCPoint1[29885] = {X 185.1830, Y 7.3639, Z -2.1667, A 0.000, B 0.000, C 0.000 }
gfCNCPoint1[29886] = {X 187.5576, Y 7.3679, Z -2.1667, A 0.000, B 0.000, C 0.000 }
gfCNCPoint1[29887] = {X 189.9199, Y 7.6105, Z -2.1667, A 0.000, B 0.000, C 0.000 }
gfCNCPoint1[29888] = {X 191.6609, Y 7.9688, Z -2.1667, A 0.000, B 0.000, C 0.000 }
gfCNCPoint1[29889] = {X 193.3561, Y 8.5038, Z -2.1667, A 0.000, B 0.000, C 0.000 }
gfCNCPoint1[29890] = {X 194.9873, Y 9.2101, Z -2.1667, A 0.000, B 0.000, C 0.000 }
gfCNCPoint1[29891] = {X 196.5375, Y 10.0800, Z -2.1667, A 0.000, B 0.000, C 0.000 }
gfCNCPoint1[29892] = {X 197.9902, Y 11.1043, Z -2.1667, A 0.000, B 0.000, C 0.000 }
gfCNCPoint1[29893] = {X 199.2816, Y 12.2863, Z -2.1667, A 0.000, B 0.000, C 0.000 }
gfCNCPoint1[29894] = {X 200.4010, Y 13.6322, Z -2.1667, A 0.000, B 0.000, C 0.000 }
gfCNCPoint1[29895] = {X 201.3278, Y 15.1175, Z -2.1667, A 0.000, B 0.000, C 0.000 }
gfCNCPoint1[29896] = {X 202.0447, Y 16.7146, Z -2.1667, A 0.000, B 0.000, C 0.000 }
gfCNCPoint1[29897] = {X 202.5135, Y 18.3531, Z -2.1667, A 0.000, B 0.000, C 0.000 }
gfCNCPoint1[29898] = {X 202.7918, Y 20.0344, Z -2.1667, A 0.000, B 0.000, C 0.000 }
gfCNCPoint1[29899] = {X 202.8757, Y 21.7366, Z -2.1667, A 0.000, B 0.000, C 0.000 }
gfCNCPoint1[29900] = {X 202.7642, Y 23.4371, Z -2.1667, A 0.000, B 0.000, C 0.000 }
gfCNCPoint1[29901] = {X 202.4588, Y 25.1138, Z -2.1667, A 0.000, B 0.000, C 0.000 }
gfCNCPoint1[29902] = {X 202.0010, Y 26.5984, Z -2.1667, A 0.000, B 0.000, C 0.000 }
gfCNCPoint1[29903] = {X 201.3477, Y 28.0081, Z -2.1667, A 0.000, B 0.000, C 0.000 }
gfCNCPoint1[29904] = {X 200.5108, Y 29.3171, Z -2.1667, A 0.000, B 0.000, C 0.000 }
gfCNCPoint1[29905] = {X 199.5056, Y 30.5017, Z -2.1667, A 0.000, B 0.000, C 0.000 }
gfCNCPoint1[29906] = {X 198.3502, Y 31.5405, Z -2.1667, A 0.000, B 0.000, C 0.000 }
gfCNCPoint1[29907] = {X 199.2140, Y 31.8437, Z -2.1667, A 0.000, B 0.000, C 0.000 }
gfCNCPoint1[29908] = {X 199.9905, Y 32.3285, Z -2.1667, A 0.000, B 0.000, C 0.000 }
gfCNCPoint1[29909] = {X 200.6422, Y 32.9715, Z -2.1667, A 0.000, B 0.000, C 0.000 }
gfCNCPoint1[29910] = {X 201.1375, Y 33.7414, Z -2.1667, A 0.000, B 0.000, C 0.000 }
gfCNCPoint1[29911] = {X 204.1781, Y 40.0227, Z -2.1667, A 0.000, B 0.000, C 0.000 }
gfCNCPoint1[29912] = {X 204.4868, Y 40.8982, Z -2.1667, A 0.000, B 0.000, C 0.000 }
gfCNCPoint1[29913] = {X 204.5937, Y 41.8203, Z -2.1667, A 0.000, B 0.000, C 0.000 }
gfCNCPoint1[29914] = {X 204.4934, Y 42.7431, Z -2.1667, A 0.000, B 0.000, C 0.000 }
gfCNCPoint1[29915] = {X 204.1910, Y 43.6208, Z -2.1667, A 0.000, B 0.000, C 0.000 }
gfCNCPoint1[29916] = {X 203.7015, Y 44.4095, Z -2.1667, A 0.000, B 0.000, C 0.000 }
gfCNCPoint1[29917] = {X 203.0493, Y 45.0700, Z -2.1667, A 0.000, B 0.000, C 0.000 }
gfCNCPoint1[29918] = {X 202.5130, Y 45.5036, Z -2.1667, A 0.000, B 0.000, C 0.000 }
gfCNCPoint1[29919] = {X 201.8221, Y 45.9562, Z -2.1667, A 0.000, B 0.000, C 0.000 }
gfCNCPoint1[29920] = {X 201.0556, Y 46.2639, Z -2.1667, A 0.000, B 0.000, C 0.000 }
gfCNCPoint1[29921] = {X 200.2435, Y 46.4147, Z -2.1667, A 0.000, B 0.000, C 0.000 }
gfCNCPoint1[29922] = {X 199.4176, Y 46.4028, Z -2.1667, A 0.000, B 0.000, C 0.000 }
gfCNCPoint1[29923] = {X 198.6102, Y 46.2285, Z -2.1667, A 0.000, B 0.000, C 0.000 }
gfCNCPoint1[29924] = {X 196.8690, Y 47.1575, Z -2.1667, A 0.000, B 0.000, C 0.000 }
gfCNCPoint1[29925] = {X 195.0676, Y 47.9636, Z -2.1667, A 0.000, B 0.000, C 0.000 }
gfCNCPoint1[29926] = {X 193.2147, Y 48.6431, Z -2.1667, A 0.000, B 0.000, C 0.000 }
gfCNCPoint1[29927] = {X 191.3192, Y 49.1926, Z -2.1667, A 0.000, B 0.000, C 0.000 }
gfCNCPoint1[29928] = {X 189.3899, Y 49.5835, Z -2.1667, A 0.000, B 0.000, C 0.000 }
gfCNCPoint1[29929] = {X 187.4337, Y 49.8042, Z -2.1667, A 0.000, B 0.000, C 0.000 }
gfCNCPoint1[29930] = {X 185.4658, Y 49.8529, Z -2.1667, A 0.000, B 0.000, C 0.000 }
gfCNCPoint1[29931] = {X 183.5011, Y 49.7294, Z -2.1667, A 0.000, B 0.000, C 0.000 }
gfCNCPoint1[29932] = {X 181.5548, Y 49.4346, Z -2.1667, A 0.000, B 0.000, C 0.000 }
gfCNCPoint1[29933] = {X 179.6859, Y 48.9675, Z -2.1667, A 0.000, B 0.000, C 0.000 }
gfCNCPoint1[29934] = {X 177.8824, Y 48.2904, Z -2.1667, A 0.000, B 0.000, C 0.000 }
gfCNCPoint1[29935] = {X 176.1678, Y 47.4122, Z -2.1667, A 0.000, B 0.000, C 0.000 }
gfCNCPoint1[29936] = {X 174.5645, Y 46.3442, Z -2.1667, A 0.000, B 0.000, C 0.000 }
gfCNCPoint1[29937] = {X 173.3463, Y 45.3161, Z -2.1667, A 0.000, B 0.000, C 0.000 }
gfCNCPoint1[29938] = {X 172.2624, Y 44.1474, Z -2.1667, A 0.000, B 0.000, C 0.000 }
gfCNCPoint1[29939] = {X 171.3287, Y 42.8554, Z -2.1667, A 0.000, B 0.000, C 0.000 }
gfCNCPoint1[29940] = {X 170.5592, Y 41.4595, Z -2.1667, A 0.000, B 0.000, C 0.000 }
gfCNCPoint1[29941] = {X 169.9653, Y 39.9802, Z -2.1667, A 0.000, B 0.000, C 0.000 }
gfCNCPoint1[29942] = {X 169.5559, Y 38.4397, Z -2.1667, A 0.000, B 0.000, C 0.000 }
gfCNCPoint1[29943] = {X 169.3369, Y 36.8608, Z -2.1667, A 0.000, B 0.000, C 0.000 }
gfCNCPoint1[29944] = {X 169.2533, Y 35.0463, Z -2.1667, A 0.000, B 0.000, C 0.000 }
gfCNCPoint1[29945] = {X 169.3976, Y 33.2356, Z -2.1667, A 0.000, B 0.000, C 0.000 }
gfCNCPoint1[29946] = {X 169.7677, Y 31.4572, Z -2.1667, A 0.000, B 0.000, C 0.000 }
gfCNCPoint1[29947] = {X 170.3575, Y 29.7393, Z -2.1667, A 0.000, B 0.000, C 0.000 }
gfCNCPoint1[29948] = {X 171.0243, Y 28.3873, Z -2.1667, A 0.000, B 0.000, C 0.000 }
gfCNCPoint1[29949] = {X 171.8744, Y 27.1424, Z -2.1667, A 0.000, B 0.000, C 0.000 }
gfCNCPoint1[29950] = {X 172.8909, Y 26.0292, Z -2.1667, A 0.000, B 0.000, C 0.000 }
gfCNCPoint1[29951] = {X 174.0537, Y 25.0699, Z -2.1667, A 0.000, B 0.000, C 0.000 }
gfCNCPoint1[29952] = {X 175.3398, Y 24.2835, Z -2.1667, A 0.000, B 0.000, C 0.000 }
gfCNCPoint1[29953] = {X 174.4753, Y 23.9355, Z -2.1667, A 0.000, B 0.000, C 0.000 }
gfCNCPoint1[29954] = {X 173.7100, Y 23.4038, Z -2.1667, A 0.000, B 0.000, C 0.000 }
gfCNCPoint1[29955] = {X 173.0822, Y 22.7151, Z -2.1667, A 0.000, B 0.000, C 0.000 }
gfCNCPoint1[29956] = {X 172.6235, Y 21.9039, Z -2.1667, A 0.000, B 0.000, C 0.000 }
gfCNCPoint1[29957] = {X 171.3062, Y 18.6783, Z -2.1667, A 0.000, B 0.000, C 0.000 }
gfCNCPoint1[29958] = {X 167.6031, Y 20.1905, Z -2.1667, A 0.000, B 0.000, C 0.000 }
gfCNCPoint1[29959] = {X 171.3803, Y 18.6480, Z -2.1667, A 0.000, B 0.000, C 0.000 }
gfCNCPoint1[29960] = {X 170.0626, Y 15.4213, Z -2.1667, A 0.000, B 0.000, C 0.000 }
gfCNCPoint1[29961] = {X 169.8043, Y 14.4793, Z -2.1667, A 0.000, B 0.000, C 0.000 }
gfCNCPoint1[29962] = {X 169.7773, Y 13.5028, Z -2.1667, A 0.000, B 0.000, C 0.000 }
gfCNCPoint1[29963] = {X 169.9832, Y 12.5479, Z -2.1667, A 0.000, B 0.000, C 0.000 }
gfCNCPoint1[29964] = {X 170.4102, Y 11.6694, Z -2.1667, A 0.000, B 0.000, C 0.000 }
gfCNCPoint1[29965] = {X 171.0337, Y 10.9174, Z -2.1667, A 0.000, B 0.000, C 0.000 }
gfCNCPoint1[29966] = {X 171.8181, Y 10.3353, Z -2.1667, A 0.000, B 0.000, C 0.000 }
gfCNCPoint1[29967] = {X 172.4475, Y 9.9764, Z -2.1667, A 0.000, B 0.000, C 0.000 }
gfCNCPoint1[29968] = {X 173.3053, Y 9.6186, Z -2.1667, A 0.000, B 0.000, C 0.000 }
gfCNCPoint1[29969] = {X 174.2218, Y 9.4641, Z -2.1667, A 0.000, B 0.000, C 0.000 }
gfCNCPoint1[29970] = {X 175.1494, Y 9.5211, Z -2.1667, A 0.000, B 0.000, C 0.000 }
gfCNCPoint1[29971] = {X 176.0401, Y 9.7866, Z -2.1667, A 0.000, B 0.000, C 0.000 }
gfCNCPoint1[29972] = {X 178.2232, Y 8.8574, Z -2.1667, A 0.000, B 0.000, C 0.000 }
gfCNCPoint1[29973] = {X 180.4889, Y 8.1530, Z -2.1667, A 0.000, B 0.000, C 0.000 }
gfCNCPoint1[29974] = {X 182.8140, Y 7.6803, Z -2.1667, A 0.000, B 0.000, C 0.000 }
gfCNCPoint1[29975] = {X 185.1748, Y 7.4444, Z -2.1667, A 0.000, B 0.000, C 0.000 }
gfCNCPoint1[29976] = {X 187.5475, Y 7.4474, Z -2.1667, A 0.000, B 0.000, C 0.000 }
gfCNCPoint1[29977] = {X 189.9077, Y 7.6895, Z -2.1667, A 0.000, B 0.000, C 0.000 }
gfCNCPoint1[29978] = {X 191.6407, Y 8.0462, Z -2.1667, A 0.000, B 0.000, C 0.000 }
gfCNCPoint1[29979] = {X 193.3280, Y 8.5788, Z -2.1667, A 0.000, B 0.000, C 0.000 }
gfCNCPoint1[29980] = {X 194.9518, Y 9.2817, Z -2.1667, A 0.000, B 0.000, C 0.000 }
gfCNCPoint1[29981] = {X 196.4948, Y 10.1476, Z -2.1667, A 0.000, B 0.000, C 0.000 }
gfCNCPoint1[29982] = {X 197.9408, Y 11.1673, Z -2.1667, A 0.000, B 0.000, C 0.000 }
gfCNCPoint1[29983] = {X 199.2239, Y 12.3417, Z -2.1667, A 0.000, B 0.000, C 0.000 }
gfCNCPoint1[29984] = {X 200.3362, Y 13.6791, Z -2.1667, A 0.000, B 0.000, C 0.000 }
gfCNCPoint1[29985] = {X 201.2570, Y 15.1548, Z -2.1667, A 0.000, B 0.000, C 0.000 }
gfCNCPoint1[29986] = {X 201.9694, Y 16.7417, Z -2.1667, A 0.000, B 0.000, C 0.000 }
